Yaskawa INFORM job: A_NAIHAN_0617_1_PAINT_3.JBI

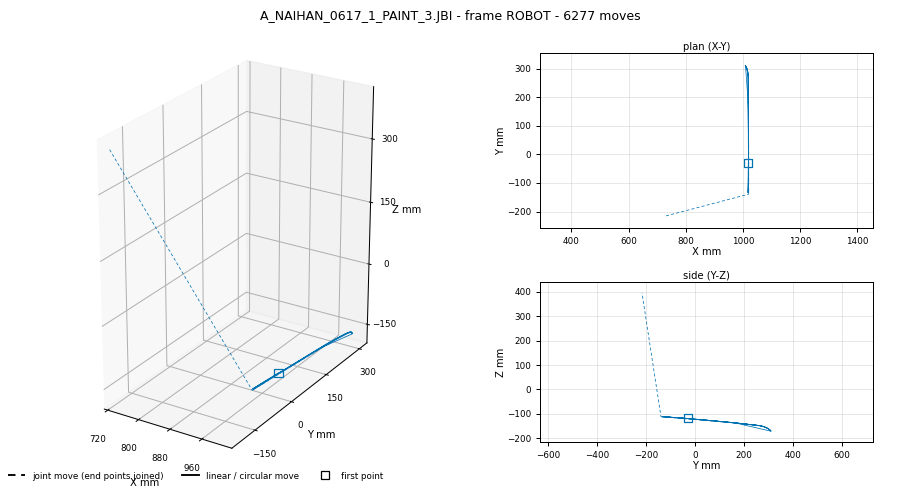
[picture p0: tool path of A_NAIHAN_0617_1_PAINT_3.JBI in frame ROBOT, 6277 of 6277 moves have a stored position in this frame; points joined in program order, loops and branches not executed]
/JOB
//NAME A_NAIHAN_0617_1_PAINT3
//POS
///NPOS 6277,0,0,0,0,0
///TOOL 1
///USER 0
///POSTYPE ROBOT
///RECTAN
///RCONF 0,0,0,0,1,0,0,0,0,0,0,0,0,0,0,0,0,0,0,0,0,0,0,0
C00000=1018.547,-30.236,-118.214,-24.117,21.565,-43.265
C00001=1018.547,-30.633,-118.183,-24.117,21.566,-43.271
C00002=1018.546,-31.031,-118.151,-24.116,21.567,-43.277
C00003=1018.545,-31.428,-118.119,-24.115,21.568,-43.282
C00004=1018.545,-31.825,-118.086,-24.114,21.567,-43.287
C00005=1018.543,-32.223,-118.054,-24.114,21.568,-43.293
C00006=1018.543,-32.621,-118.022,-24.113,21.569,-43.299
C00007=1018.542,-33.018,-117.990,-24.112,21.570,-43.304
C00008=1018.541,-33.415,-117.958,-24.111,21.570,-43.310
C00009=1018.540,-33.812,-117.926,-24.111,21.570,-43.315
C00010=1018.539,-34.210,-117.894,-24.110,21.571,-43.321
C00011=1018.539,-34.608,-117.863,-24.109,21.571,-43.328
C00012=1018.538,-35.005,-117.831,-24.108,21.572,-43.334
C00013=1018.536,-35.402,-117.799,-24.107,21.572,-43.339
C00014=1018.535,-35.799,-117.767,-24.107,21.573,-43.344
C00015=1018.535,-36.197,-117.735,-24.106,21.573,-43.350
C00016=1018.533,-36.594,-117.703,-24.105,21.574,-43.356
C00017=1018.532,-36.992,-117.671,-24.105,21.575,-43.361
C00018=1018.531,-37.389,-117.640,-24.104,21.575,-43.366
C00019=1018.530,-37.786,-117.608,-24.103,21.576,-43.372
C00020=1018.529,-38.183,-117.577,-24.102,21.576,-43.378
C00021=1018.528,-38.581,-117.544,-24.102,21.577,-43.383
C00022=1018.527,-38.978,-117.513,-24.101,21.578,-43.389
C00023=1018.526,-39.375,-117.481,-24.100,21.578,-43.394
C00024=1018.524,-39.772,-117.450,-24.099,21.579,-43.400
C00025=1018.524,-40.170,-117.418,-24.099,21.579,-43.405
C00026=1018.522,-40.567,-117.387,-24.098,21.580,-43.411
C00027=1018.520,-40.965,-117.355,-24.097,21.581,-43.417
C00028=1018.519,-41.362,-117.323,-24.096,21.582,-43.422
C00029=1018.518,-41.760,-117.292,-24.096,21.582,-43.427
C00030=1018.517,-42.156,-117.260,-24.095,21.582,-43.433
C00031=1018.515,-42.553,-117.228,-24.094,21.583,-43.439
C00032=1018.514,-42.951,-117.198,-24.093,21.584,-43.444
C00033=1018.513,-43.348,-117.166,-24.092,21.584,-43.451
C00034=1018.512,-43.745,-117.134,-24.092,21.585,-43.457
C00035=1018.511,-44.143,-117.103,-24.091,21.585,-43.462
C00036=1018.509,-44.540,-117.071,-24.090,21.585,-43.468
C00037=1018.508,-44.937,-117.040,-24.089,21.586,-43.473
C00038=1018.506,-45.334,-117.009,-24.089,21.587,-43.479
C00039=1018.505,-45.731,-116.977,-24.088,21.588,-43.485
C00040=1018.503,-46.128,-116.946,-24.087,21.589,-43.490
C00041=1018.501,-46.525,-116.915,-24.086,21.588,-43.496
C00042=1018.499,-46.923,-116.883,-24.086,21.589,-43.501
C00043=1018.498,-47.320,-116.853,-24.085,21.590,-43.507
C00044=1018.497,-47.717,-116.821,-24.084,21.591,-43.512
C00045=1018.496,-47.937,-116.804,-24.084,21.591,-43.516
C00046=1018.495,-48.156,-116.786,-24.083,21.591,-43.520
C00047=1018.493,-48.511,-116.759,-24.083,21.592,-43.525
C00048=1018.492,-48.908,-116.728,-24.082,21.592,-43.531
C00049=1018.490,-49.305,-116.696,-24.081,21.592,-43.536
C00050=1018.488,-49.703,-116.666,-24.080,21.593,-43.542
C00051=1018.487,-50.099,-116.634,-24.080,21.594,-43.547
C00052=1018.485,-50.496,-116.603,-24.079,21.595,-43.553
C00053=1018.483,-50.894,-116.572,-24.078,21.595,-43.558
C00054=1018.482,-51.291,-116.541,-24.077,21.596,-43.564
C00055=1018.479,-51.687,-116.510,-24.077,21.597,-43.570
C00056=1018.478,-52.085,-116.479,-24.076,21.598,-43.575
C00057=1018.477,-52.481,-116.448,-24.075,21.598,-43.581
C00058=1018.474,-52.877,-116.417,-24.074,21.598,-43.588
C00059=1018.473,-53.275,-116.386,-24.073,21.599,-43.593
C00060=1018.471,-53.671,-116.355,-24.073,21.599,-43.599
C00061=1018.469,-54.068,-116.324,-24.072,21.600,-43.604
C00062=1018.467,-54.466,-116.293,-24.071,21.601,-43.610
C00063=1018.465,-54.862,-116.262,-24.071,21.602,-43.616
C00064=1018.463,-55.259,-116.232,-24.070,21.603,-43.621
C00065=1018.461,-55.657,-116.200,-24.069,21.602,-43.627
C00066=1018.459,-56.054,-116.170,-24.068,21.603,-43.632
C00067=1018.457,-56.452,-116.139,-24.067,21.603,-43.639
C00068=1018.455,-56.850,-116.108,-24.067,21.604,-43.645
C00069=1018.452,-57.248,-116.077,-24.066,21.605,-43.651
C00070=1018.451,-57.647,-116.047,-24.065,21.606,-43.656
C00071=1018.449,-58.047,-116.016,-24.064,21.606,-43.662
C00072=1018.447,-58.447,-115.985,-24.064,21.607,-43.667
C00073=1018.445,-58.846,-115.954,-24.063,21.608,-43.673
C00074=1018.443,-59.247,-115.923,-24.062,21.608,-43.680
C00075=1018.441,-59.648,-115.892,-24.061,21.609,-43.686
C00076=1018.438,-60.050,-115.861,-24.061,21.610,-43.691
C00077=1018.436,-60.453,-115.831,-24.060,21.610,-43.697
C00078=1018.434,-60.856,-115.799,-24.059,21.610,-43.702
C00079=1018.431,-61.260,-115.768,-24.058,21.611,-43.708
C00080=1018.429,-61.663,-115.737,-24.057,21.611,-43.715
C00081=1018.427,-62.068,-115.705,-24.057,21.612,-43.720
C00082=1018.424,-62.473,-115.675,-24.056,21.613,-43.726
C00083=1018.421,-62.879,-115.643,-24.055,21.614,-43.732
C00084=1018.419,-63.285,-115.612,-24.054,21.615,-43.737
C00085=1018.417,-63.691,-115.581,-24.053,21.615,-43.744
C00086=1018.415,-64.099,-115.550,-24.053,21.615,-43.750
C00087=1018.412,-64.506,-115.519,-24.052,21.616,-43.756
C00088=1018.409,-64.915,-115.487,-24.051,21.617,-43.761
C00089=1018.407,-65.323,-115.457,-24.050,21.617,-43.768
C00090=1018.404,-65.732,-115.425,-24.049,21.618,-43.774
C00091=1018.402,-66.142,-115.394,-24.049,21.619,-43.780
C00092=1018.399,-66.551,-115.362,-24.048,21.620,-43.785
C00093=1018.396,-66.961,-115.331,-24.047,21.620,-43.791
C00094=1018.393,-67.371,-115.300,-24.046,21.621,-43.798
C00095=1018.391,-67.781,-115.269,-24.046,21.621,-43.804
C00096=1018.388,-68.191,-115.238,-24.045,21.622,-43.809
C00097=1018.385,-68.601,-115.206,-24.044,21.623,-43.815
C00098=1018.382,-69.013,-115.175,-24.043,21.623,-43.822
C00099=1018.380,-69.423,-115.144,-24.042,21.624,-43.827
C00100=1018.377,-69.834,-115.113,-24.042,21.625,-43.833
C00101=1018.374,-70.245,-115.082,-24.041,21.625,-43.839
C00102=1018.371,-70.656,-115.050,-24.040,21.626,-43.846
C00103=1018.368,-71.067,-115.019,-24.039,21.626,-43.851
C00104=1018.365,-71.478,-114.989,-24.039,21.627,-43.857
C00105=1018.362,-71.888,-114.957,-24.038,21.628,-43.865
C00106=1018.359,-72.299,-114.926,-24.037,21.629,-43.870
C00107=1018.356,-72.710,-114.895,-24.036,21.630,-43.876
C00108=1018.353,-73.121,-114.864,-24.035,21.631,-43.881
C00109=1018.350,-73.532,-114.833,-24.034,21.631,-43.888
C00110=1018.348,-73.942,-114.803,-24.034,21.632,-43.894
C00111=1018.344,-74.353,-114.771,-24.033,21.632,-43.900
C00112=1018.341,-74.763,-114.740,-24.032,21.633,-43.905
C00113=1018.338,-75.173,-114.710,-24.031,21.633,-43.912
C00114=1018.335,-75.583,-114.679,-24.031,21.634,-43.918
C00115=1018.331,-75.993,-114.648,-24.030,21.635,-43.924
C00116=1018.329,-76.402,-114.617,-24.029,21.636,-43.929
C00117=1018.326,-76.810,-114.586,-24.028,21.636,-43.936
C00118=1018.321,-77.220,-114.556,-24.027,21.637,-43.942
C00119=1018.319,-77.628,-114.525,-24.027,21.637,-43.948
C00120=1018.315,-78.036,-114.494,-24.026,21.638,-43.953
C00121=1018.312,-78.443,-114.464,-24.025,21.638,-43.960
C00122=1018.309,-78.851,-114.434,-24.024,21.639,-43.966
C00123=1018.305,-79.257,-114.403,-24.023,21.640,-43.972
C00124=1018.302,-79.663,-114.373,-24.023,21.641,-43.977
C00125=1018.299,-80.069,-114.342,-24.022,21.641,-43.984
C00126=1018.295,-80.474,-114.313,-24.021,21.642,-43.990
C00127=1018.292,-80.878,-114.283,-24.020,21.643,-43.995
C00128=1018.288,-81.283,-114.252,-24.020,21.643,-44.001
C00129=1018.285,-81.686,-114.222,-24.019,21.644,-44.007
C00130=1018.281,-82.089,-114.192,-24.018,21.644,-44.014
C00131=1018.278,-82.490,-114.162,-24.017,21.645,-44.019
C00132=1018.274,-82.892,-114.133,-24.016,21.646,-44.025
C00133=1018.271,-83.293,-114.103,-24.016,21.647,-44.031
C00134=1018.267,-83.693,-114.073,-24.015,21.648,-44.036
C00135=1018.264,-84.093,-114.043,-24.014,21.648,-44.043
C00136=1018.260,-84.499,-114.013,-24.013,21.649,-44.049
C00137=1018.258,-84.723,-113.996,-24.013,21.649,-44.053
C00138=1018.256,-84.964,-113.979,-24.012,21.650,-44.056
C00139=1018.254,-85.218,-113.959,-24.012,21.649,-44.060
C00140=1018.251,-85.472,-113.941,-24.012,21.650,-44.062
C00141=1018.248,-85.718,-113.923,-24.011,21.650,-44.065
C00142=1018.246,-85.948,-113.905,-24.011,21.651,-44.069
C00143=1018.243,-86.357,-113.875,-24.010,21.652,-44.077
C00144=1018.239,-86.745,-113.846,-24.009,21.652,-44.082
C00145=1018.236,-87.125,-113.818,-24.008,21.652,-44.087
C00146=1018.232,-87.497,-113.791,-24.007,21.653,-44.093
C00147=1018.228,-87.869,-113.764,-24.007,21.654,-44.099
C00148=1018.225,-88.244,-113.736,-24.006,21.655,-44.104
C00149=1018.221,-88.652,-113.706,-24.005,21.656,-44.112
C00150=1018.218,-88.899,-113.688,-24.005,21.656,-44.116
C00151=1018.216,-89.174,-113.668,-24.004,21.657,-44.117
C00152=1018.213,-89.458,-113.646,-24.004,21.656,-44.121
C00153=1018.210,-89.733,-113.626,-24.003,21.657,-44.124
C00154=1018.208,-89.983,-113.607,-24.003,21.657,-44.128
C00155=1018.205,-90.202,-113.591,-24.002,21.658,-44.132
C00156=1018.201,-90.598,-113.563,-24.002,21.659,-44.138
C00157=1018.198,-90.992,-113.534,-24.001,21.659,-44.145
C00158=1018.194,-91.384,-113.505,-24.000,21.660,-44.150
C00159=1018.190,-91.776,-113.476,-23.999,21.660,-44.156
C00160=1018.186,-92.168,-113.447,-23.999,21.661,-44.162
C00161=1018.182,-92.558,-113.419,-23.998,21.662,-44.167
C00162=1018.178,-92.948,-113.390,-23.997,21.663,-44.173
C00163=1018.174,-93.338,-113.362,-23.996,21.664,-44.178
C00164=1018.170,-93.726,-113.333,-23.996,21.664,-44.184
C00165=1018.166,-94.113,-113.305,-23.995,21.664,-44.189
C00166=1018.162,-94.500,-113.277,-23.994,21.665,-44.195
C00167=1018.157,-94.886,-113.248,-23.994,21.666,-44.200
C00168=1018.153,-95.272,-113.220,-23.993,21.666,-44.207
C00169=1018.149,-95.657,-113.192,-23.992,21.667,-44.213
C00170=1018.145,-96.041,-113.164,-23.991,21.668,-44.219
C00171=1018.141,-96.425,-113.136,-23.990,21.668,-44.224
C00172=1018.136,-96.809,-113.109,-23.990,21.669,-44.230
C00173=1018.132,-97.193,-113.081,-23.989,21.669,-44.235
C00174=1018.127,-97.576,-113.053,-23.988,21.670,-44.241
C00175=1018.124,-97.959,-113.025,-23.988,21.671,-44.246
C00176=1018.119,-98.342,-112.997,-23.987,21.672,-44.252
C00177=1018.116,-98.726,-112.969,-23.986,21.673,-44.258
C00178=1018.111,-99.109,-112.941,-23.985,21.673,-44.263
C00179=1018.106,-99.493,-112.914,-23.985,21.673,-44.268
C00180=1018.102,-99.877,-112.885,-23.984,21.674,-44.274
C00181=1018.097,-100.261,-112.857,-23.983,21.675,-44.280
C00182=1018.093,-100.647,-112.830,-23.982,21.676,-44.285
C00183=1018.089,-101.032,-112.802,-23.982,21.677,-44.291
C00184=1018.084,-101.418,-112.774,-23.981,21.676,-44.296
C00185=1018.079,-101.806,-112.746,-23.980,21.677,-44.302
C00186=1018.075,-102.194,-112.718,-23.980,21.678,-44.307
C00187=1018.070,-102.582,-112.690,-23.979,21.678,-44.314
C00188=1018.065,-102.971,-112.661,-23.978,21.679,-44.320
C00189=1018.060,-103.361,-112.634,-23.977,21.680,-44.326
C00190=1018.056,-103.751,-112.606,-23.976,21.681,-44.331
C00191=1018.051,-104.143,-112.577,-23.976,21.682,-44.337
C00192=1018.046,-104.535,-112.549,-23.975,21.681,-44.342
C00193=1018.041,-104.926,-112.521,-23.974,21.682,-44.348
C00194=1018.037,-105.318,-112.492,-23.974,21.683,-44.353
C00195=1018.032,-105.711,-112.464,-23.973,21.684,-44.359
C00196=1018.027,-106.104,-112.436,-23.972,21.685,-44.365
C00197=1018.022,-106.497,-112.408,-23.971,21.686,-44.370
C00198=1018.017,-106.890,-112.380,-23.971,21.686,-44.376
C00199=1018.012,-107.283,-112.352,-23.970,21.687,-44.383
C00200=1018.006,-107.675,-112.323,-23.969,21.687,-44.388
C00201=1018.002,-108.068,-112.295,-23.968,21.688,-44.394
C00202=1017.997,-108.461,-112.267,-23.968,21.688,-44.399
C00203=1017.992,-108.854,-112.239,-23.967,21.689,-44.405
C00204=1017.986,-109.247,-112.211,-23.966,21.690,-44.411
C00205=1017.981,-109.639,-112.183,-23.965,21.691,-44.416
C00206=1017.976,-110.032,-112.155,-23.965,21.691,-44.422
C00207=1017.971,-110.425,-112.127,-23.964,21.692,-44.427
C00208=1017.966,-110.818,-112.099,-23.963,21.693,-44.433
C00209=1017.961,-111.211,-112.071,-23.963,21.694,-44.439
C00210=1017.954,-111.603,-112.043,-23.962,21.694,-44.446
C00211=1017.949,-111.996,-112.015,-23.961,21.694,-44.451
C00212=1017.944,-112.389,-111.987,-23.960,21.695,-44.456
C00213=1017.938,-112.781,-111.958,-23.959,21.696,-44.462
C00214=1017.933,-113.174,-111.930,-23.959,21.696,-44.468
C00215=1017.927,-113.567,-111.903,-23.958,21.697,-44.473
C00216=1017.922,-113.959,-111.874,-23.957,21.698,-44.479
C00217=1017.916,-114.352,-111.847,-23.957,21.699,-44.485
C00218=1017.911,-114.745,-111.819,-23.956,21.700,-44.490
C00219=1017.906,-115.136,-111.791,-23.955,21.701,-44.496
C00220=1017.900,-115.529,-111.764,-23.954,21.700,-44.501
C00221=1017.894,-115.921,-111.735,-23.954,21.701,-44.507
C00222=1017.889,-116.314,-111.708,-23.953,21.702,-44.512
C00223=1017.883,-116.706,-111.680,-23.952,21.703,-44.518
C00224=1017.877,-117.099,-111.652,-23.952,21.704,-44.523
C00225=1017.872,-117.492,-111.624,-23.951,21.705,-44.529
C00226=1017.866,-117.883,-111.596,-23.950,21.705,-44.536
C00227=1017.860,-118.276,-111.569,-23.949,21.705,-44.541
C00228=1017.854,-118.668,-111.541,-23.948,21.706,-44.547
C00229=1017.849,-119.060,-111.513,-23.948,21.706,-44.553
C00230=1017.842,-119.452,-111.485,-23.947,21.707,-44.558
C00231=1017.837,-119.845,-111.458,-23.946,21.708,-44.564
C00232=1017.831,-120.237,-111.430,-23.946,21.709,-44.569
C00233=1017.824,-120.628,-111.403,-23.945,21.710,-44.575
C00234=1017.819,-121.021,-111.375,-23.944,21.710,-44.580
C00235=1017.812,-121.413,-111.347,-23.943,21.710,-44.586
C00236=1017.807,-121.805,-111.320,-23.943,21.711,-44.591
C00237=1017.800,-122.197,-111.292,-23.942,21.712,-44.597
C00238=1017.794,-122.590,-111.265,-23.941,21.713,-44.603
C00239=1017.788,-122.982,-111.237,-23.941,21.714,-44.608
C00240=1017.782,-123.373,-111.209,-23.940,21.715,-44.614
C00241=1017.776,-123.766,-111.182,-23.939,21.714,-44.619
C00242=1017.770,-124.158,-111.154,-23.939,21.715,-44.625
C00243=1017.763,-124.549,-111.126,-23.938,21.716,-44.630
C00244=1017.757,-124.942,-111.099,-23.937,21.717,-44.636
C00245=1017.750,-125.334,-111.072,-23.936,21.718,-44.642
C00246=1017.743,-125.725,-111.044,-23.936,21.719,-44.647
C00247=1017.738,-126.117,-111.017,-23.935,21.719,-44.652
C00248=1017.731,-126.509,-110.989,-23.934,21.719,-44.658
C00249=1017.725,-126.901,-110.962,-23.934,21.720,-44.664
C00250=1017.719,-127.294,-110.934,-23.933,21.721,-44.669
C00251=1017.712,-127.685,-110.907,-23.932,21.722,-44.675
C00252=1017.705,-128.077,-110.879,-23.932,21.723,-44.680
C00253=1017.699,-128.469,-110.853,-23.931,21.723,-44.686
C00254=1017.692,-128.861,-110.825,-23.930,21.723,-44.691
C00255=1017.685,-129.253,-110.798,-23.929,21.724,-44.697
C00256=1017.679,-129.644,-110.770,-23.929,21.725,-44.703
C00257=1017.672,-130.036,-110.744,-23.928,21.726,-44.708
C00258=1017.665,-130.428,-110.716,-23.927,21.727,-44.714
C00259=1017.658,-130.820,-110.689,-23.926,21.727,-44.719
C00260=1017.652,-131.211,-110.661,-23.926,21.728,-44.725
C00261=1017.645,-131.604,-110.634,-23.925,21.728,-44.730
C00262=1017.638,-131.995,-110.607,-23.924,21.729,-44.736
C00263=1017.631,-132.387,-110.579,-23.924,21.730,-44.741
C00264=1017.625,-132.779,-110.552,-23.923,21.730,-44.747
C00265=1017.618,-133.171,-110.524,-23.922,21.731,-44.752
C00266=1017.610,-133.563,-110.498,-23.922,21.732,-44.758
C00267=1017.604,-133.954,-110.470,-23.921,21.732,-44.763
C00268=1017.988,-133.926,-110.710,-23.921,21.732,-44.763
C00269=1017.995,-133.535,-110.737,-23.922,21.732,-44.758
C00270=1018.002,-133.143,-110.765,-23.922,21.731,-44.752
C00271=1018.008,-132.751,-110.792,-23.923,21.730,-44.747
C00272=1018.015,-132.360,-110.818,-23.924,21.730,-44.741
C00273=1018.022,-131.968,-110.846,-23.924,21.729,-44.736
C00274=1018.029,-131.576,-110.872,-23.925,21.728,-44.730
C00275=1018.035,-131.184,-110.900,-23.926,21.728,-44.725
C00276=1018.042,-130.792,-110.928,-23.926,21.727,-44.719
C00277=1018.049,-130.400,-110.954,-23.927,21.727,-44.714
C00278=1018.055,-130.009,-110.982,-23.928,21.726,-44.708
C00279=1018.062,-129.617,-111.009,-23.929,21.725,-44.703
C00280=1018.068,-129.225,-111.036,-23.929,21.724,-44.697
C00281=1018.075,-128.833,-111.064,-23.930,21.723,-44.691
C00282=1018.081,-128.441,-111.091,-23.931,21.723,-44.686
C00283=1018.087,-128.050,-111.118,-23.932,21.723,-44.680
C00284=1018.094,-127.658,-111.145,-23.932,21.722,-44.675
C00285=1018.101,-127.265,-111.172,-23.933,21.721,-44.669
C00286=1018.107,-126.873,-111.200,-23.934,21.720,-44.664
C00287=1018.113,-126.482,-111.227,-23.934,21.719,-44.658
C00288=1018.120,-126.090,-111.254,-23.935,21.719,-44.652
C00289=1018.126,-125.698,-111.283,-23.936,21.719,-44.647
C00290=1018.132,-125.306,-111.309,-23.936,21.718,-44.642
C00291=1018.138,-124.914,-111.337,-23.937,21.717,-44.636
C00292=1018.144,-124.522,-111.364,-23.938,21.716,-44.630
C00293=1018.150,-124.130,-111.392,-23.939,21.715,-44.625
C00294=1018.157,-123.738,-111.419,-23.939,21.714,-44.619
C00295=1018.162,-123.346,-111.447,-23.940,21.715,-44.614
C00296=1018.168,-122.954,-111.474,-23.941,21.714,-44.608
C00297=1018.175,-122.562,-111.502,-23.941,21.713,-44.603
C00298=1018.180,-122.170,-111.529,-23.942,21.712,-44.597
C00299=1018.186,-121.778,-111.557,-23.943,21.711,-44.591
C00300=1018.192,-121.385,-111.584,-23.943,21.710,-44.586
C00301=1018.198,-120.993,-111.612,-23.944,21.710,-44.580
C00302=1018.204,-120.602,-111.639,-23.945,21.710,-44.575
C00303=1018.210,-120.210,-111.667,-23.946,21.709,-44.569
C00304=1018.216,-119.817,-111.694,-23.946,21.708,-44.564
C00305=1018.222,-119.425,-111.722,-23.947,21.707,-44.558
C00306=1018.227,-119.033,-111.749,-23.948,21.706,-44.553
C00307=1018.233,-118.641,-111.777,-23.948,21.706,-44.547
C00308=1018.239,-118.248,-111.805,-23.949,21.705,-44.541
C00309=1018.244,-117.855,-111.833,-23.950,21.705,-44.536
C00310=1018.250,-117.464,-111.861,-23.951,21.705,-44.529
C00311=1018.256,-117.071,-111.888,-23.952,21.704,-44.523
C00312=1018.261,-116.679,-111.915,-23.952,21.703,-44.518
C00313=1018.267,-116.287,-111.944,-23.953,21.702,-44.512
C00314=1018.272,-115.894,-111.971,-23.954,21.701,-44.507
C00315=1018.278,-115.502,-111.999,-23.954,21.700,-44.501
C00316=1018.284,-115.110,-112.027,-23.955,21.701,-44.496
C00317=1018.289,-114.717,-112.055,-23.956,21.700,-44.490
C00318=1018.294,-114.325,-112.082,-23.957,21.699,-44.485
C00319=1018.299,-113.932,-112.110,-23.957,21.698,-44.479
C00320=1018.305,-113.540,-112.138,-23.958,21.697,-44.473
C00321=1018.310,-113.147,-112.166,-23.959,21.696,-44.468
C00322=1018.316,-112.755,-112.194,-23.959,21.696,-44.462
C00323=1018.321,-112.362,-112.222,-23.960,21.695,-44.456
C00324=1018.326,-111.969,-112.250,-23.961,21.694,-44.451
C00325=1018.332,-111.577,-112.277,-23.962,21.694,-44.446
C00326=1018.337,-111.184,-112.305,-23.963,21.694,-44.439
C00327=1018.342,-110.791,-112.334,-23.963,21.693,-44.433
C00328=1018.347,-110.398,-112.362,-23.964,21.692,-44.427
C00329=1018.352,-110.005,-112.390,-23.965,21.691,-44.422
C00330=1018.357,-109.612,-112.418,-23.965,21.691,-44.416
C00331=1018.362,-109.219,-112.446,-23.966,21.690,-44.411
C00332=1018.367,-108.827,-112.473,-23.967,21.689,-44.405
C00333=1018.372,-108.434,-112.501,-23.968,21.688,-44.399
C00334=1018.377,-108.041,-112.529,-23.968,21.688,-44.394
C00335=1018.382,-107.649,-112.558,-23.969,21.687,-44.388
C00336=1018.387,-107.256,-112.586,-23.970,21.687,-44.383
C00337=1018.392,-106.863,-112.614,-23.971,21.686,-44.376
C00338=1018.397,-106.470,-112.642,-23.971,21.686,-44.370
C00339=1018.402,-106.077,-112.670,-23.972,21.685,-44.365
C00340=1018.407,-105.684,-112.699,-23.973,21.684,-44.359
C00341=1018.412,-105.291,-112.727,-23.974,21.683,-44.353
C00342=1018.417,-104.899,-112.755,-23.974,21.682,-44.348
C00343=1018.421,-104.507,-112.783,-23.975,21.681,-44.342
C00344=1018.426,-104.115,-112.811,-23.976,21.682,-44.337
C00345=1018.430,-103.724,-112.839,-23.976,21.681,-44.331
C00346=1018.435,-103.334,-112.867,-23.977,21.680,-44.326
C00347=1018.440,-102.944,-112.895,-23.978,21.679,-44.320
C00348=1018.444,-102.555,-112.924,-23.979,21.678,-44.314
C00349=1018.449,-102.167,-112.952,-23.980,21.678,-44.307
C00350=1018.454,-101.779,-112.979,-23.980,21.677,-44.302
C00351=1018.458,-101.391,-113.007,-23.981,21.676,-44.296
C00352=1018.463,-101.005,-113.035,-23.982,21.677,-44.291
C00353=1018.467,-100.620,-113.063,-23.982,21.676,-44.285
C00354=1018.471,-100.234,-113.091,-23.983,21.675,-44.280
C00355=1018.476,-99.849,-113.119,-23.984,21.674,-44.274
C00356=1018.480,-99.465,-113.146,-23.985,21.673,-44.268
C00357=1018.485,-99.082,-113.175,-23.985,21.673,-44.263
C00358=1018.489,-98.699,-113.202,-23.986,21.673,-44.258
C00359=1018.493,-98.315,-113.230,-23.987,21.672,-44.252
C00360=1018.497,-97.932,-113.258,-23.988,21.671,-44.246
C00361=1018.500,-97.617,-113.280,-23.988,21.670,-44.241
C00362=1018.503,-97.391,-113.297,-23.988,21.670,-44.239
C00363=1018.505,-97.166,-113.313,-23.989,21.669,-44.235
C00364=1018.510,-96.782,-113.342,-23.990,21.669,-44.230
C00365=1018.514,-96.398,-113.369,-23.990,21.668,-44.224
C00366=1018.518,-96.014,-113.397,-23.991,21.668,-44.219
C00367=1018.522,-95.630,-113.424,-23.992,21.667,-44.213
C00368=1018.526,-95.245,-113.453,-23.993,21.666,-44.207
C00369=1018.530,-94.860,-113.481,-23.994,21.666,-44.200
C00370=1018.534,-94.473,-113.510,-23.994,21.665,-44.195
C00371=1018.539,-94.086,-113.537,-23.995,21.664,-44.189
C00372=1018.543,-93.698,-113.566,-23.996,21.664,-44.184
C00373=1018.547,-93.310,-113.594,-23.996,21.664,-44.178
C00374=1018.551,-92.921,-113.623,-23.997,21.663,-44.173
C00375=1018.555,-92.531,-113.651,-23.998,21.662,-44.167
C00376=1018.558,-92.140,-113.680,-23.999,21.661,-44.162
C00377=1018.562,-91.749,-113.708,-23.999,21.660,-44.156
C00378=1018.566,-91.357,-113.737,-24.000,21.660,-44.150
C00379=1018.570,-90.964,-113.766,-24.001,21.659,-44.145
C00380=1018.574,-90.570,-113.794,-24.002,21.659,-44.138
C00381=1018.578,-90.174,-113.824,-24.002,21.658,-44.132
C00382=1018.580,-89.956,-113.840,-24.003,21.657,-44.128
C00383=1018.582,-89.706,-113.858,-24.003,21.657,-44.124
C00384=1018.585,-89.431,-113.879,-24.004,21.656,-44.121
C00385=1018.588,-89.147,-113.900,-24.004,21.657,-44.117
C00386=1018.591,-88.872,-113.919,-24.005,21.656,-44.116
C00387=1018.592,-88.625,-113.938,-24.005,21.656,-44.112
C00388=1018.597,-88.218,-113.968,-24.006,21.655,-44.104
C00389=1018.600,-87.842,-113.996,-24.007,21.654,-44.099
C00390=1018.603,-87.470,-114.023,-24.007,21.653,-44.093
C00391=1018.607,-87.098,-114.050,-24.008,21.652,-44.087
C00392=1018.610,-86.719,-114.078,-24.009,21.652,-44.082
C00393=1018.614,-86.330,-114.107,-24.010,21.652,-44.077
C00394=1018.618,-85.921,-114.137,-24.011,21.651,-44.069
C00395=1018.620,-85.691,-114.154,-24.011,21.650,-44.065
C00396=1018.622,-85.445,-114.172,-24.012,21.650,-44.062
C00397=1018.625,-85.190,-114.191,-24.012,21.649,-44.060
C00398=1018.627,-84.937,-114.210,-24.012,21.650,-44.056
C00399=1018.629,-84.696,-114.228,-24.013,21.649,-44.053
C00400=1018.631,-84.472,-114.244,-24.013,21.649,-44.049
C00401=1018.635,-84.066,-114.275,-24.014,21.648,-44.043
C00402=1018.638,-83.666,-114.303,-24.015,21.648,-44.036
C00403=1018.642,-83.266,-114.333,-24.016,21.647,-44.031
C00404=1018.645,-82.865,-114.363,-24.016,21.646,-44.025
C00405=1018.648,-82.464,-114.394,-24.017,21.645,-44.019
C00406=1018.652,-82.062,-114.423,-24.018,21.644,-44.014
C00407=1018.656,-81.659,-114.453,-24.019,21.644,-44.007
C00408=1018.659,-81.256,-114.483,-24.020,21.643,-44.001
C00409=1018.662,-80.851,-114.513,-24.020,21.643,-43.995
C00410=1018.665,-80.448,-114.543,-24.021,21.642,-43.990
C00411=1018.669,-80.042,-114.573,-24.022,21.641,-43.984
C00412=1018.673,-79.637,-114.604,-24.023,21.641,-43.977
C00413=1018.675,-79.230,-114.634,-24.023,21.640,-43.972
C00414=1018.679,-78.824,-114.664,-24.024,21.639,-43.966
C00415=1018.682,-78.417,-114.695,-24.025,21.638,-43.960
C00416=1018.685,-78.009,-114.725,-24.026,21.638,-43.953
C00417=1018.689,-77.601,-114.756,-24.027,21.637,-43.948
C00418=1018.692,-77.193,-114.787,-24.027,21.637,-43.942
C00419=1018.695,-76.784,-114.817,-24.028,21.636,-43.936
C00420=1018.698,-76.375,-114.848,-24.029,21.636,-43.929
C00421=1018.702,-75.966,-114.879,-24.030,21.635,-43.924
C00422=1018.705,-75.557,-114.909,-24.031,21.634,-43.918
C00423=1018.707,-75.146,-114.940,-24.031,21.633,-43.912
C00424=1018.711,-74.736,-114.971,-24.032,21.633,-43.905
C00425=1018.714,-74.326,-115.002,-24.033,21.632,-43.900
C00426=1018.717,-73.915,-115.032,-24.034,21.632,-43.894
C00427=1018.720,-73.505,-115.064,-24.034,21.631,-43.888
C00428=1018.723,-73.095,-115.094,-24.035,21.631,-43.881
C00429=1018.726,-72.683,-115.125,-24.036,21.630,-43.876
C00430=1018.729,-72.273,-115.157,-24.037,21.629,-43.870
C00431=1018.732,-71.862,-115.187,-24.038,21.628,-43.865
C00432=1018.735,-71.451,-115.218,-24.039,21.627,-43.857
C00433=1018.738,-71.041,-115.250,-24.039,21.626,-43.851
C00434=1018.741,-70.629,-115.281,-24.040,21.626,-43.846
C00435=1018.743,-70.218,-115.312,-24.041,21.625,-43.839
C00436=1018.746,-69.807,-115.343,-24.042,21.625,-43.833
C00437=1018.749,-69.397,-115.374,-24.042,21.624,-43.827
C00438=1018.752,-68.986,-115.405,-24.043,21.623,-43.822
C00439=1018.755,-68.576,-115.437,-24.044,21.623,-43.815
C00440=1018.757,-68.164,-115.468,-24.045,21.622,-43.809
C00441=1018.760,-67.754,-115.499,-24.046,21.621,-43.804
C00442=1018.763,-67.344,-115.531,-24.046,21.621,-43.798
C00443=1018.764,-66.934,-115.561,-24.047,21.620,-43.791
C00444=1018.767,-66.524,-115.592,-24.048,21.620,-43.785
C00445=1018.770,-66.115,-115.624,-24.049,21.619,-43.780
C00446=1018.773,-65.705,-115.655,-24.049,21.618,-43.774
C00447=1018.776,-65.297,-115.686,-24.050,21.617,-43.768
C00448=1018.778,-64.888,-115.717,-24.051,21.617,-43.761
C00449=1018.780,-64.480,-115.749,-24.052,21.616,-43.756
C00450=1018.783,-64.073,-115.780,-24.053,21.615,-43.750
C00451=1018.785,-63.666,-115.810,-24.053,21.615,-43.744
C00452=1018.787,-63.258,-115.842,-24.054,21.615,-43.737
C00453=1018.790,-62.852,-115.873,-24.055,21.614,-43.732
C00454=1018.793,-62.447,-115.904,-24.056,21.613,-43.726
C00455=1018.795,-62.041,-115.935,-24.057,21.612,-43.720
C00456=1018.796,-61.637,-115.966,-24.057,21.611,-43.715
C00457=1018.800,-61.233,-115.998,-24.058,21.611,-43.708
C00458=1018.802,-60.829,-116.028,-24.059,21.610,-43.702
C00459=1018.804,-60.426,-116.059,-24.060,21.610,-43.697
C00460=1018.806,-60.024,-116.091,-24.061,21.610,-43.691
C00461=1018.808,-59.622,-116.121,-24.061,21.609,-43.686
C00462=1018.810,-59.221,-116.152,-24.062,21.608,-43.680
C00463=1018.812,-58.820,-116.184,-24.063,21.608,-43.673
C00464=1018.815,-58.419,-116.214,-24.064,21.607,-43.667
C00465=1018.817,-58.020,-116.245,-24.064,21.606,-43.662
C00466=1018.818,-57.621,-116.276,-24.065,21.606,-43.656
C00467=1018.821,-57.222,-116.307,-24.066,21.605,-43.651
C00468=1018.823,-56.824,-116.338,-24.067,21.604,-43.645
C00469=1018.825,-56.425,-116.369,-24.067,21.603,-43.639
C00470=1018.827,-56.028,-116.399,-24.068,21.603,-43.632
C00471=1018.829,-55.630,-116.430,-24.069,21.602,-43.627
C00472=1018.831,-55.233,-116.461,-24.070,21.603,-43.621
C00473=1018.833,-54.836,-116.492,-24.071,21.602,-43.616
C00474=1018.835,-54.439,-116.522,-24.071,21.601,-43.610
C00475=1018.836,-54.042,-116.554,-24.072,21.600,-43.604
C00476=1018.838,-53.645,-116.584,-24.073,21.599,-43.599
C00477=1018.841,-53.248,-116.615,-24.073,21.599,-43.593
C00478=1018.842,-52.851,-116.647,-24.074,21.598,-43.588
C00479=1018.844,-52.454,-116.677,-24.075,21.598,-43.581
C00480=1018.846,-52.057,-116.708,-24.076,21.598,-43.575
C00481=1018.847,-51.661,-116.739,-24.077,21.597,-43.570
C00482=1018.849,-51.264,-116.770,-24.077,21.596,-43.564
C00483=1018.851,-50.867,-116.801,-24.078,21.595,-43.558
C00484=1018.853,-50.470,-116.832,-24.079,21.595,-43.553
C00485=1018.854,-50.073,-116.863,-24.080,21.594,-43.547
C00486=1018.856,-49.676,-116.895,-24.080,21.593,-43.542
C00487=1018.858,-49.279,-116.925,-24.081,21.592,-43.536
C00488=1018.859,-48.882,-116.956,-24.082,21.592,-43.531
C00489=1018.861,-48.485,-116.988,-24.083,21.592,-43.525
C00490=1018.862,-48.087,-117.019,-24.084,21.592,-43.518
C00491=1018.864,-47.691,-117.050,-24.084,21.591,-43.512
C00492=1018.866,-47.294,-117.081,-24.085,21.590,-43.507
C00493=1018.867,-46.896,-117.112,-24.086,21.589,-43.501
C00494=1018.868,-46.499,-117.144,-24.086,21.588,-43.496
C00495=1018.869,-46.102,-117.175,-24.087,21.589,-43.490
C00496=1018.871,-45.705,-117.206,-24.088,21.588,-43.485
C00497=1018.872,-45.308,-117.238,-24.089,21.587,-43.479
C00498=1018.874,-44.910,-117.269,-24.089,21.586,-43.473
C00499=1018.875,-44.513,-117.300,-24.090,21.585,-43.468
C00500=1018.877,-44.116,-117.332,-24.091,21.585,-43.462
C00501=1018.878,-43.718,-117.363,-24.092,21.585,-43.457
C00502=1018.880,-43.321,-117.395,-24.092,21.584,-43.451
C00503=1018.881,-42.924,-117.426,-24.093,21.584,-43.444
C00504=1018.883,-42.527,-117.457,-24.094,21.583,-43.439
C00505=1018.884,-42.130,-117.489,-24.095,21.582,-43.433
C00506=1018.885,-41.733,-117.521,-24.096,21.582,-43.427
C00507=1018.886,-41.335,-117.552,-24.096,21.582,-43.422
C00508=1018.888,-40.938,-117.584,-24.097,21.581,-43.417
C00509=1018.889,-40.541,-117.615,-24.098,21.580,-43.411
C00510=1018.890,-40.143,-117.647,-24.099,21.579,-43.405
C00511=1018.891,-39.746,-117.678,-24.099,21.579,-43.400
C00512=1018.892,-39.349,-117.710,-24.100,21.578,-43.394
C00513=1018.893,-38.952,-117.741,-24.101,21.578,-43.389
C00514=1018.895,-38.555,-117.773,-24.102,21.577,-43.383
C00515=1018.895,-38.157,-117.805,-24.102,21.576,-43.378
C00516=1018.897,-37.760,-117.836,-24.103,21.576,-43.372
C00517=1018.898,-37.362,-117.868,-24.104,21.575,-43.366
C00518=1018.900,-36.965,-117.900,-24.105,21.575,-43.361
C00519=1018.900,-36.568,-117.932,-24.105,21.574,-43.356
C00520=1018.901,-36.170,-117.964,-24.106,21.573,-43.350
C00521=1018.902,-35.773,-117.995,-24.107,21.573,-43.344
C00522=1018.903,-35.376,-118.027,-24.107,21.572,-43.339
C00523=1018.903,-34.978,-118.059,-24.108,21.572,-43.334
C00524=1018.905,-34.581,-118.091,-24.109,21.571,-43.328
C00525=1018.906,-34.184,-118.123,-24.110,21.571,-43.321
C00526=1018.907,-33.786,-118.155,-24.111,21.570,-43.315
C00527=1018.907,-33.389,-118.186,-24.111,21.570,-43.310
C00528=1018.908,-32.991,-118.219,-24.112,21.570,-43.304
C00529=1018.909,-32.594,-118.251,-24.113,21.569,-43.299
C00530=1018.911,-32.196,-118.283,-24.114,21.568,-43.293
C00531=1018.911,-31.799,-118.315,-24.114,21.567,-43.287
C00532=1018.912,-31.401,-118.346,-24.115,21.568,-43.282
C00533=1018.913,-31.004,-118.379,-24.116,21.567,-43.277
C00534=1018.913,-30.607,-118.411,-24.117,21.566,-43.271
C00535=1018.914,-30.210,-118.443,-24.117,21.565,-43.265
C00536=1018.915,-29.812,-118.475,-24.118,21.565,-43.260
C00537=1018.915,-29.415,-118.507,-24.119,21.565,-43.255
C00538=1018.915,-29.017,-118.539,-24.120,21.564,-43.249
C00539=1018.916,-28.620,-118.572,-24.120,21.563,-43.243
C00540=1018.917,-28.222,-118.604,-24.121,21.562,-43.238
C00541=1018.918,-27.825,-118.636,-24.122,21.562,-43.232
C00542=1018.919,-27.427,-118.668,-24.123,21.562,-43.227
C00543=1018.920,-27.030,-118.701,-24.123,21.561,-43.221
C00544=1018.920,-26.632,-118.733,-24.124,21.560,-43.217
C00545=1018.920,-26.235,-118.765,-24.125,21.560,-43.212
C00546=1018.921,-25.837,-118.797,-24.125,21.559,-43.206
C00547=1018.921,-25.440,-118.830,-24.126,21.558,-43.201
C00548=1018.922,-25.043,-118.862,-24.127,21.558,-43.195
C00549=1018.923,-24.645,-118.894,-24.128,21.558,-43.190
C00550=1018.923,-24.248,-118.927,-24.128,21.557,-43.184
C00551=1018.924,-23.851,-118.959,-24.129,21.556,-43.178
C00552=1018.924,-23.453,-118.992,-24.130,21.556,-43.173
C00553=1018.924,-23.055,-119.023,-24.131,21.555,-43.168
C00554=1018.924,-22.658,-119.056,-24.131,21.555,-43.162
C00555=1018.925,-22.260,-119.088,-24.132,21.554,-43.156
C00556=1018.925,-21.862,-119.122,-24.133,21.554,-43.151
C00557=1018.926,-21.464,-119.154,-24.134,21.553,-43.146
C00558=1018.926,-21.067,-119.186,-24.134,21.552,-43.140
C00559=1018.926,-20.670,-119.219,-24.135,21.553,-43.135
C00560=1018.926,-20.272,-119.252,-24.136,21.552,-43.129
C00561=1018.927,-19.875,-119.284,-24.136,21.551,-43.123
C00562=1018.927,-19.464,-119.318,-24.138,21.551,-43.116
C00563=1018.927,-19.215,-119.339,-24.138,21.550,-43.113
C00564=1018.927,-18.926,-119.363,-24.139,21.550,-43.109
C00565=1018.928,-18.615,-119.388,-24.139,21.550,-43.107
C00566=1018.927,-18.304,-119.414,-24.139,21.549,-43.105
C00567=1018.928,-18.016,-119.437,-24.139,21.549,-43.101
C00568=1018.928,-17.768,-119.458,-24.140,21.548,-43.098
C00569=1018.929,-17.357,-119.492,-24.141,21.547,-43.090
C00570=1018.929,-16.960,-119.524,-24.142,21.548,-43.085
C00571=1018.929,-16.561,-119.556,-24.142,21.547,-43.079
C00572=1018.928,-16.163,-119.590,-24.143,21.546,-43.074
C00573=1018.929,-15.763,-119.623,-24.144,21.546,-43.068
C00574=1018.928,-15.362,-119.656,-24.145,21.545,-43.063
C00575=1018.929,-14.959,-119.689,-24.145,21.545,-43.057
C00576=1018.929,-14.554,-119.723,-24.146,21.544,-43.052
C00577=1018.929,-14.146,-119.757,-24.147,21.544,-43.046
C00578=1018.929,-13.734,-119.791,-24.148,21.543,-43.041
C00579=1018.929,-13.320,-119.825,-24.148,21.543,-43.035
C00580=1018.929,-12.902,-119.860,-24.149,21.542,-43.029
C00581=1018.929,-12.483,-119.895,-24.150,21.542,-43.024
C00582=1018.929,-12.272,-119.912,-24.150,21.541,-43.022
C00583=1018.929,-12.060,-119.930,-24.151,21.541,-43.019
C00584=1018.929,-11.848,-119.947,-24.151,21.540,-43.016
C00585=1018.928,-11.637,-119.965,-24.151,21.540,-43.013
C00586=1018.928,-11.424,-119.983,-24.152,21.540,-43.011
C00587=1018.929,-11.210,-120.001,-24.152,21.540,-43.007
C00588=1018.928,-10.996,-120.018,-24.152,21.539,-43.006
C00589=1018.929,-10.783,-120.036,-24.153,21.539,-43.002
C00590=1018.929,-10.567,-120.054,-24.153,21.539,-42.998
C00591=1018.929,-10.353,-120.072,-24.154,21.538,-42.996
C00592=1018.928,-10.137,-120.090,-24.154,21.539,-42.993
C00593=1018.928,-9.921,-120.108,-24.154,21.538,-42.991
C00594=1018.928,-9.706,-120.125,-24.155,21.538,-42.987
C00595=1018.928,-9.490,-120.143,-24.155,21.538,-42.985
C00596=1018.928,-9.273,-120.162,-24.156,21.537,-42.982
C00597=1018.928,-9.057,-120.180,-24.156,21.537,-42.980
C00598=1018.928,-8.841,-120.198,-24.156,21.536,-42.976
C00599=1018.928,-8.624,-120.216,-24.157,21.537,-42.973
C00600=1018.928,-8.407,-120.234,-24.157,21.536,-42.971
C00601=1018.927,-8.191,-120.252,-24.158,21.536,-42.967
C00602=1018.927,-7.974,-120.270,-24.158,21.536,-42.965
C00603=1018.928,-7.756,-120.288,-24.158,21.535,-42.961
C00604=1018.927,-7.538,-120.306,-24.159,21.535,-42.959
C00605=1018.927,-7.319,-120.325,-24.159,21.534,-42.956
C00606=1018.927,-7.099,-120.343,-24.160,21.535,-42.952
C00607=1018.927,-6.877,-120.362,-24.160,21.534,-42.950
C00608=1018.927,-6.655,-120.380,-24.160,21.534,-42.947
C00609=1018.926,-6.432,-120.399,-24.161,21.533,-42.944
C00610=1018.927,-6.208,-120.418,-24.161,21.533,-42.941
C00611=1018.926,-5.983,-120.436,-24.161,21.533,-42.939
C00612=1018.926,-5.760,-120.455,-24.162,21.533,-42.935
C00613=1018.925,-5.535,-120.475,-24.162,21.532,-42.934
C00614=1018.926,-5.312,-120.493,-24.163,21.532,-42.930
C00615=1018.925,-5.089,-120.512,-24.163,21.532,-42.927
C00616=1018.925,-4.868,-120.530,-24.163,21.532,-42.925
C00617=1018.924,-4.648,-120.549,-24.164,21.531,-42.921
C00618=1018.924,-4.429,-120.567,-24.164,21.531,-42.919
C00619=1018.924,-4.213,-120.585,-24.165,21.531,-42.915
C00620=1018.924,-3.997,-120.603,-24.165,21.530,-42.913
C00621=1018.924,-3.784,-120.621,-24.165,21.530,-42.910
C00622=1018.924,-3.571,-120.639,-24.166,21.530,-42.908
C00623=1018.923,-3.360,-120.657,-24.166,21.530,-42.904
C00624=1018.923,-2.939,-120.692,-24.167,21.529,-42.899
C00625=1018.922,-2.520,-120.728,-24.168,21.529,-42.893
C00626=1018.922,-2.102,-120.763,-24.169,21.529,-42.888
C00627=1018.922,-1.687,-120.797,-24.169,21.528,-42.882
C00628=1018.921,-1.274,-120.832,-24.170,21.527,-42.877
C00629=1018.920,-0.865,-120.867,-24.171,21.527,-42.872
C00630=1018.920,-0.456,-120.901,-24.171,21.526,-42.867
C00631=1018.920,-0.051,-120.936,-24.172,21.525,-42.862
C00632=1018.919,0.352,-120.970,-24.173,21.525,-42.857
C00633=1018.918,0.754,-121.004,-24.173,21.525,-42.851
C00634=1018.918,1.155,-121.038,-24.174,21.525,-42.846
C00635=1018.917,1.552,-121.071,-24.175,21.523,-42.841
C00636=1018.917,1.951,-121.105,-24.175,21.524,-42.836
C00637=1018.916,2.337,-121.138,-24.176,21.523,-42.833
C00638=1018.915,2.689,-121.168,-24.177,21.522,-42.827
C00639=1018.915,3.012,-121.195,-24.177,21.522,-42.823
C00640=1018.915,3.326,-121.221,-24.178,21.521,-42.817
C00641=1018.914,3.654,-121.249,-24.179,21.521,-42.812
C00642=1018.913,4.013,-121.280,-24.179,21.521,-42.809
C00643=1018.912,4.402,-121.313,-24.180,21.520,-42.805
C00644=1018.911,4.798,-121.347,-24.180,21.519,-42.799
C00645=1018.910,5.194,-121.380,-24.181,21.520,-42.794
C00646=1018.910,5.589,-121.413,-24.182,21.519,-42.790
C00647=1018.909,5.983,-121.448,-24.182,21.518,-42.785
C00648=1018.909,6.376,-121.481,-24.183,21.519,-42.779
C00649=1018.907,6.769,-121.515,-24.184,21.517,-42.775
C00650=1018.907,7.162,-121.548,-24.185,21.517,-42.770
C00651=1018.906,7.552,-121.582,-24.185,21.517,-42.764
C00652=1018.905,7.940,-121.614,-24.186,21.516,-42.761
C00653=1018.904,8.324,-121.647,-24.187,21.516,-42.755
C00654=1018.903,8.705,-121.680,-24.187,21.515,-42.751
C00655=1018.902,9.083,-121.712,-24.188,21.515,-42.746
C00656=1018.901,9.459,-121.744,-24.189,21.514,-42.740
C00657=1018.900,9.835,-121.776,-24.189,21.514,-42.737
C00658=1018.899,10.211,-121.809,-24.190,21.513,-42.731
C00659=1018.899,10.590,-121.841,-24.191,21.513,-42.726
C00660=1018.898,10.970,-121.874,-24.191,21.513,-42.722
C00661=1018.896,11.354,-121.907,-24.192,21.512,-42.716
C00662=1018.895,11.739,-121.940,-24.192,21.511,-42.713
C00663=1018.895,12.126,-121.973,-24.193,21.512,-42.707
C00664=1018.893,12.512,-122.006,-24.193,21.510,-42.703
C00665=1018.893,12.898,-122.039,-24.194,21.510,-42.698
C00666=1018.892,13.285,-122.073,-24.195,21.511,-42.693
C00667=1018.890,13.672,-122.106,-24.196,21.509,-42.689
C00668=1018.889,14.059,-122.140,-24.196,21.509,-42.683
C00669=1018.888,14.447,-122.173,-24.197,21.509,-42.680
C00670=1018.887,14.835,-122.206,-24.198,21.508,-42.674
C00671=1018.886,15.224,-122.240,-24.198,21.508,-42.670
C00672=1018.885,15.614,-122.273,-24.199,21.507,-42.665
C00673=1018.883,16.004,-122.307,-24.200,21.507,-42.659
C00674=1018.882,16.395,-122.341,-24.200,21.506,-42.656
C00675=1018.881,16.787,-122.375,-24.201,21.506,-42.650
C00676=1018.880,17.179,-122.409,-24.201,21.505,-42.646
C00677=1018.879,17.572,-122.442,-24.202,21.505,-42.641
C00678=1018.877,17.967,-122.476,-24.203,21.505,-42.635
C00679=1018.876,18.362,-122.511,-24.203,21.504,-42.632
C00680=1018.875,18.758,-122.545,-24.204,21.503,-42.626
C00681=1018.873,19.154,-122.580,-24.205,21.503,-42.622
C00682=1018.872,19.552,-122.614,-24.205,21.503,-42.617
C00683=1018.871,19.763,-122.632,-24.206,21.503,-42.613
C00684=1018.870,19.999,-122.652,-24.206,21.502,-42.610
C00685=1018.870,20.264,-122.675,-24.207,21.503,-42.606
C00686=1018.868,20.552,-122.700,-24.207,21.501,-42.604
C00687=1018.867,20.848,-122.726,-24.207,21.501,-42.602
C00688=1018.867,21.140,-122.752,-24.208,21.502,-42.599
C00689=1018.866,21.412,-122.775,-24.208,21.501,-42.597
C00690=1018.865,21.657,-122.797,-24.209,21.501,-42.593
C00691=1018.863,22.070,-122.833,-24.210,21.501,-42.586
C00692=1018.862,22.445,-122.865,-24.210,21.500,-42.584
C00693=1018.860,22.767,-122.893,-24.211,21.500,-42.580
C00694=1018.860,23.033,-122.916,-24.211,21.500,-42.577
C00695=1018.859,23.265,-122.936,-24.211,21.499,-42.573
C00696=1018.858,23.499,-122.957,-24.212,21.498,-42.567
C00697=1018.858,23.771,-122.981,-24.213,21.498,-42.564
C00698=1018.855,24.101,-123.010,-24.213,21.498,-42.562
C00699=1018.854,24.485,-123.043,-24.213,21.497,-42.558
C00700=1018.853,24.884,-123.078,-24.214,21.497,-42.553
C00701=1018.851,25.283,-123.113,-24.215,21.497,-42.549
C00702=1018.849,25.683,-123.147,-24.215,21.496,-42.543
C00703=1018.848,26.082,-123.182,-24.216,21.496,-42.540
C00704=1018.846,26.482,-123.217,-24.217,21.496,-42.534
C00705=1018.845,26.881,-123.252,-24.218,21.495,-42.529
C00706=1018.843,27.280,-123.287,-24.218,21.494,-42.525
C00707=1018.841,27.679,-123.322,-24.219,21.495,-42.520
C00708=1018.840,28.078,-123.357,-24.219,21.493,-42.516
C00709=1018.838,28.478,-123.393,-24.220,21.493,-42.510
C00710=1018.837,28.878,-123.428,-24.221,21.493,-42.507
C00711=1018.835,29.278,-123.462,-24.221,21.492,-42.501
C00712=1018.833,29.677,-123.497,-24.222,21.492,-42.497
C00713=1018.831,30.076,-123.533,-24.223,21.492,-42.492
C00714=1018.829,30.476,-123.567,-24.223,21.491,-42.488
C00715=1018.828,30.876,-123.603,-24.224,21.491,-42.483
C00716=1018.826,31.275,-123.638,-24.224,21.490,-42.479
C00717=1018.824,31.674,-123.673,-24.225,21.490,-42.474
C00718=1018.822,32.075,-123.708,-24.226,21.489,-42.469
C00719=1018.820,32.474,-123.743,-24.226,21.489,-42.464
C00720=1018.818,32.874,-123.779,-24.227,21.489,-42.461
C00721=1018.817,33.273,-123.814,-24.228,21.489,-42.455
C00722=1018.814,33.673,-123.849,-24.228,21.487,-42.451
C00723=1018.813,34.073,-123.885,-24.229,21.488,-42.446
C00724=1018.811,34.473,-123.919,-24.229,21.487,-42.442
C00725=1018.808,34.872,-123.955,-24.230,21.486,-42.437
C00726=1018.807,35.272,-123.990,-24.231,21.486,-42.433
C00727=1018.805,35.672,-124.026,-24.231,21.486,-42.428
C00728=1018.803,36.071,-124.061,-24.232,21.486,-42.424
C00729=1018.801,36.471,-124.096,-24.233,21.485,-42.418
C00730=1018.799,36.871,-124.131,-24.233,21.484,-42.414
C00731=1018.797,37.271,-124.167,-24.234,21.485,-42.409
C00732=1018.795,37.670,-124.202,-24.235,21.484,-42.405
C00733=1018.793,38.071,-124.238,-24.235,21.483,-42.400
C00734=1018.790,38.470,-124.274,-24.236,21.483,-42.396
C00735=1018.789,38.871,-124.308,-24.237,21.483,-42.391
C00736=1018.787,39.270,-124.344,-24.237,21.483,-42.387
C00737=1018.785,39.670,-124.379,-24.238,21.482,-42.383
C00738=1018.783,40.070,-124.415,-24.238,21.481,-42.378
C00739=1018.780,40.470,-124.451,-24.239,21.481,-42.374
C00740=1018.778,40.869,-124.486,-24.240,21.481,-42.369
C00741=1018.776,41.270,-124.522,-24.240,21.481,-42.365
C00742=1018.773,41.670,-124.558,-24.241,21.480,-42.359
C00743=1018.771,42.070,-124.594,-24.241,21.479,-42.356
C00744=1018.769,42.470,-124.629,-24.242,21.479,-42.352
C00745=1018.767,42.870,-124.665,-24.243,21.479,-42.347
C00746=1018.765,43.270,-124.700,-24.243,21.479,-42.343
C00747=1018.762,43.670,-124.735,-24.244,21.479,-42.338
C00748=1018.760,44.070,-124.772,-24.244,21.477,-42.333
C00749=1018.758,44.470,-124.807,-24.245,21.477,-42.330
C00750=1018.756,44.870,-124.843,-24.246,21.477,-42.325
C00751=1018.753,45.269,-124.879,-24.246,21.477,-42.321
C00752=1018.751,45.671,-124.915,-24.247,21.477,-42.316
C00753=1018.748,46.070,-124.950,-24.247,21.475,-42.311
C00754=1018.747,46.470,-124.986,-24.248,21.475,-42.308
C00755=1018.744,46.870,-125.022,-24.249,21.475,-42.302
C00756=1018.742,47.271,-125.058,-24.249,21.475,-42.299
C00757=1018.738,47.671,-125.093,-24.250,21.474,-42.295
C00758=1018.736,48.071,-125.129,-24.251,21.474,-42.290
C00759=1018.734,48.471,-125.165,-24.251,21.474,-42.286
C00760=1018.731,48.871,-125.201,-24.251,21.472,-42.282
C00761=1018.729,49.271,-125.237,-24.252,21.473,-42.277
C00762=1018.727,49.671,-125.273,-24.253,21.472,-42.273
C00763=1018.724,50.072,-125.309,-24.254,21.472,-42.268
C00764=1018.721,50.471,-125.344,-24.254,21.472,-42.264
C00765=1018.719,50.872,-125.381,-24.255,21.471,-42.260
C00766=1018.716,51.272,-125.417,-24.255,21.471,-42.255
C00767=1018.714,51.672,-125.453,-24.256,21.471,-42.251
C00768=1018.711,52.072,-125.489,-24.256,21.470,-42.247
C00769=1018.709,52.473,-125.525,-24.257,21.469,-42.243
C00770=1018.706,52.872,-125.561,-24.258,21.469,-42.238
C00771=1018.704,53.273,-125.597,-24.258,21.469,-42.234
C00772=1018.700,53.673,-125.633,-24.259,21.468,-42.230
C00773=1018.697,54.073,-125.669,-24.259,21.468,-42.225
C00774=1018.695,54.473,-125.705,-24.260,21.468,-42.221
C00775=1018.693,54.873,-125.741,-24.260,21.468,-42.218
C00776=1018.690,55.274,-125.777,-24.261,21.468,-42.212
C00777=1018.687,55.673,-125.813,-24.262,21.467,-42.209
C00778=1018.685,56.074,-125.850,-24.262,21.467,-42.205
C00779=1018.682,56.474,-125.886,-24.263,21.465,-42.201
C00780=1018.679,56.875,-125.922,-24.264,21.466,-42.196
C00781=1018.676,57.275,-125.958,-24.264,21.465,-42.192
C00782=1018.673,57.675,-125.994,-24.264,21.465,-42.188
C00783=1018.670,58.075,-126.031,-24.265,21.465,-42.183
C00784=1018.667,58.475,-126.067,-24.266,21.464,-42.179
C00785=1018.665,58.876,-126.103,-24.266,21.464,-42.175
C00786=1018.662,59.276,-126.139,-24.267,21.463,-42.172
C00787=1018.659,59.676,-126.176,-24.268,21.464,-42.166
C00788=1018.656,60.076,-126.212,-24.268,21.463,-42.163
C00789=1018.653,60.476,-126.248,-24.269,21.463,-42.159
C00790=1018.651,60.876,-126.285,-24.269,21.462,-42.155
C00791=1018.647,61.276,-126.321,-24.270,21.462,-42.150
C00792=1018.644,61.677,-126.358,-24.270,21.462,-42.146
C00793=1018.641,62.077,-126.394,-24.271,21.461,-42.142
C00794=1018.638,62.477,-126.430,-24.271,21.461,-42.139
C00795=1018.635,62.896,-126.468,-24.272,21.460,-42.133
C00796=1018.633,63.150,-126.492,-24.272,21.460,-42.131
C00797=1018.631,63.417,-126.516,-24.273,21.460,-42.129
C00798=1018.629,63.667,-126.539,-24.273,21.459,-42.127
C00799=1018.628,63.885,-126.558,-24.274,21.460,-42.124
C00800=1018.626,64.092,-126.577,-24.274,21.460,-42.122
C00801=1018.625,64.310,-126.597,-24.274,21.459,-42.120
C00802=1018.623,64.538,-126.618,-24.274,21.459,-42.116
C00803=1018.621,64.775,-126.639,-24.275,21.459,-42.115
C00804=1018.619,65.011,-126.660,-24.275,21.458,-42.113
C00805=1018.617,65.241,-126.682,-24.275,21.458,-42.111
C00806=1018.615,65.462,-126.702,-24.276,21.459,-42.108
C00807=1018.614,65.675,-126.721,-24.276,21.458,-42.106
C00808=1018.611,66.083,-126.759,-24.277,21.458,-42.102
C00809=1018.607,66.481,-126.795,-24.277,21.457,-42.098
C00810=1018.605,66.881,-126.831,-24.278,21.457,-42.094
C00811=1018.601,67.284,-126.868,-24.278,21.457,-42.089
C00812=1018.598,67.687,-126.905,-24.279,21.457,-42.085
C00813=1018.595,68.092,-126.941,-24.279,21.456,-42.082
C00814=1018.592,68.498,-126.979,-24.280,21.456,-42.078
C00815=1018.589,68.906,-127.016,-24.280,21.455,-42.074
C00816=1018.585,69.314,-127.053,-24.281,21.455,-42.069
C00817=1018.582,69.724,-127.091,-24.282,21.455,-42.065
C00818=1018.578,70.135,-127.129,-24.282,21.454,-42.061
C00819=1018.575,70.547,-127.167,-24.283,21.454,-42.058
C00820=1018.572,70.958,-127.203,-24.283,21.453,-42.054
C00821=1018.568,71.369,-127.241,-24.284,21.454,-42.049
C00822=1018.564,71.780,-127.279,-24.285,21.453,-42.045
C00823=1018.561,72.192,-127.317,-24.285,21.453,-42.041
C00824=1018.557,72.606,-127.355,-24.285,21.452,-42.037
C00825=1018.555,73.021,-127.393,-24.286,21.452,-42.034
C00826=1018.550,73.439,-127.432,-24.287,21.452,-42.028
C00827=1018.547,73.859,-127.470,-24.287,21.452,-42.025
C00828=1018.545,74.071,-127.489,-24.288,21.451,-42.023
C00829=1018.544,74.283,-127.509,-24.288,21.451,-42.021
C00830=1018.542,74.495,-127.528,-24.288,21.451,-42.019
C00831=1018.540,74.708,-127.549,-24.288,21.451,-42.017
C00832=1018.538,74.922,-127.568,-24.289,21.450,-42.015
C00833=1018.536,75.136,-127.587,-24.289,21.451,-42.012
C00834=1018.534,75.349,-127.607,-24.289,21.451,-42.010
C00835=1018.532,75.561,-127.626,-24.290,21.450,-42.008
C00836=1018.528,75.981,-127.665,-24.290,21.450,-42.004
C00837=1018.525,76.393,-127.703,-24.291,21.449,-42.001
C00838=1018.522,76.795,-127.740,-24.291,21.449,-41.997
C00839=1018.518,77.190,-127.776,-24.292,21.449,-41.994
C00840=1018.514,77.578,-127.812,-24.292,21.448,-41.989
C00841=1018.511,77.964,-127.848,-24.293,21.447,-41.986
C00842=1018.508,78.351,-127.883,-24.293,21.448,-41.980
C00843=1018.504,78.741,-127.919,-24.294,21.447,-41.977
C00844=1018.501,79.139,-127.955,-24.294,21.447,-41.973
C00845=1018.497,79.543,-127.993,-24.295,21.447,-41.970
C00846=1018.493,79.958,-128.032,-24.296,21.447,-41.966
C00847=1018.491,80.169,-128.051,-24.296,21.446,-41.964
C00848=1018.489,80.380,-128.071,-24.296,21.446,-41.962
C00849=1018.488,80.593,-128.090,-24.296,21.446,-41.960
C00850=1018.486,80.805,-128.110,-24.297,21.446,-41.958
C00851=1018.483,81.019,-128.129,-24.297,21.445,-41.956
C00852=1018.481,81.232,-128.149,-24.297,21.445,-41.955
C00853=1018.480,81.444,-128.169,-24.297,21.445,-41.953
C00854=1018.477,81.657,-128.189,-24.298,21.445,-41.951
C00855=1018.475,81.869,-128.208,-24.298,21.445,-41.949
C00856=1018.473,82.080,-128.228,-24.298,21.444,-41.947
C00857=1018.472,82.292,-128.247,-24.299,21.445,-41.944
C00858=1018.470,82.503,-128.266,-24.299,21.444,-41.942
C00859=1018.467,82.714,-128.286,-24.299,21.444,-41.940
C00860=1018.466,82.924,-128.305,-24.299,21.444,-41.938
C00861=1018.462,83.345,-128.344,-24.300,21.444,-41.935
C00862=1018.458,83.763,-128.383,-24.300,21.444,-41.931
C00863=1018.454,84.181,-128.422,-24.301,21.443,-41.927
C00864=1018.450,84.596,-128.460,-24.301,21.443,-41.923
C00865=1018.446,85.011,-128.499,-24.302,21.443,-41.920
C00866=1018.442,85.423,-128.538,-24.302,21.442,-41.916
C00867=1018.438,85.834,-128.575,-24.303,21.442,-41.912
C00868=1018.434,86.243,-128.613,-24.303,21.441,-41.908
C00869=1018.429,86.650,-128.651,-24.304,21.442,-41.905
C00870=1018.426,87.055,-128.689,-24.304,21.441,-41.901
C00871=1018.422,87.459,-128.725,-24.305,21.441,-41.898
C00872=1018.419,87.855,-128.763,-24.305,21.440,-41.894
C00873=1018.415,88.243,-128.799,-24.306,21.440,-41.890
C00874=1018.410,88.626,-128.834,-24.307,21.440,-41.887
C00875=1018.407,89.009,-128.870,-24.307,21.440,-41.883
C00876=1018.403,89.396,-128.906,-24.308,21.439,-41.879
C00877=1018.399,89.789,-128.942,-24.308,21.439,-41.875
C00878=1018.395,90.187,-128.979,-24.309,21.439,-41.872
C00879=1018.390,90.586,-129.017,-24.309,21.439,-41.868
C00880=1018.387,90.986,-129.054,-24.310,21.438,-41.865
C00881=1018.383,91.385,-129.091,-24.310,21.438,-41.861
C00882=1018.379,91.783,-129.128,-24.311,21.438,-41.857
C00883=1018.374,92.183,-129.166,-24.311,21.438,-41.854
C00884=1018.370,92.582,-129.203,-24.312,21.437,-41.850
C00885=1018.366,92.982,-129.239,-24.312,21.437,-41.846
C00886=1018.362,93.380,-129.277,-24.312,21.437,-41.844
C00887=1018.358,93.779,-129.314,-24.313,21.436,-41.841
C00888=1018.354,94.178,-129.351,-24.313,21.436,-41.837
C00889=1018.349,94.578,-129.389,-24.314,21.435,-41.833
C00890=1018.345,94.977,-129.426,-24.315,21.436,-41.830
C00891=1018.341,95.376,-129.463,-24.315,21.435,-41.826
C00892=1018.337,95.774,-129.500,-24.316,21.435,-41.822
C00893=1018.332,96.173,-129.538,-24.316,21.435,-41.819
C00894=1018.328,96.572,-129.575,-24.317,21.435,-41.815
C00895=1018.324,96.971,-129.612,-24.317,21.434,-41.811
C00896=1018.319,97.370,-129.649,-24.318,21.434,-41.808
C00897=1018.315,97.769,-129.686,-24.318,21.433,-41.806
C00898=1018.311,98.167,-129.724,-24.318,21.433,-41.802
C00899=1018.307,98.566,-129.762,-24.319,21.432,-41.798
C00900=1018.303,98.965,-129.799,-24.319,21.433,-41.795
C00901=1018.298,99.364,-129.836,-24.320,21.432,-41.791
C00902=1018.294,99.763,-129.874,-24.320,21.432,-41.787
C00903=1018.289,100.162,-129.911,-24.321,21.432,-41.784
C00904=1018.284,100.560,-129.948,-24.322,21.432,-41.780
C00905=1018.280,100.959,-129.985,-24.322,21.431,-41.778
C00906=1018.276,101.358,-130.022,-24.322,21.431,-41.775
C00907=1018.271,101.757,-130.060,-24.323,21.431,-41.771
C00908=1018.267,102.155,-130.098,-24.323,21.430,-41.767
C00909=1018.262,102.555,-130.135,-24.324,21.430,-41.763
C00910=1018.258,102.953,-130.172,-24.324,21.430,-41.760
C00911=1018.253,103.352,-130.210,-24.325,21.430,-41.756
C00912=1018.249,103.750,-130.247,-24.325,21.430,-41.754
C00913=1018.244,104.149,-130.285,-24.326,21.429,-41.751
C00914=1018.240,104.548,-130.322,-24.326,21.429,-41.747
C00915=1018.235,104.946,-130.359,-24.327,21.429,-41.743
C00916=1018.231,105.345,-130.396,-24.327,21.429,-41.740
C00917=1018.226,105.744,-130.435,-24.328,21.428,-41.736
C00918=1018.221,106.142,-130.472,-24.328,21.428,-41.734
C00919=1018.217,106.541,-130.509,-24.328,21.427,-41.730
C00920=1018.212,106.940,-130.547,-24.329,21.427,-41.727
C00921=1018.207,107.338,-130.584,-24.330,21.427,-41.723
C00922=1018.203,107.737,-130.622,-24.330,21.427,-41.719
C00923=1018.198,108.136,-130.660,-24.330,21.426,-41.717
C00924=1018.193,108.534,-130.696,-24.331,21.426,-41.714
C00925=1018.188,108.933,-130.735,-24.331,21.426,-41.710
C00926=1018.184,109.332,-130.772,-24.332,21.426,-41.707
C00927=1018.179,109.730,-130.809,-24.332,21.426,-41.703
C00928=1018.174,110.128,-130.847,-24.333,21.425,-41.701
C00929=1018.169,110.527,-130.885,-24.333,21.425,-41.697
C00930=1018.164,110.926,-130.922,-24.334,21.425,-41.694
C00931=1018.160,111.323,-130.960,-24.334,21.425,-41.690
C00932=1018.155,111.722,-130.997,-24.334,21.424,-41.688
C00933=1018.150,112.122,-131.035,-24.335,21.423,-41.684
C00934=1018.145,112.520,-131.072,-24.335,21.424,-41.681
C00935=1018.140,112.919,-131.111,-24.336,21.423,-41.677
C00936=1018.135,113.317,-131.147,-24.336,21.423,-41.675
C00937=1018.131,113.716,-131.185,-24.337,21.423,-41.671
C00938=1018.125,114.114,-131.223,-24.337,21.422,-41.668
C00939=1018.121,114.513,-131.261,-24.338,21.423,-41.664
C00940=1018.115,114.911,-131.298,-24.338,21.422,-41.662
C00941=1018.111,115.310,-131.336,-24.339,21.422,-41.659
C00942=1018.105,115.708,-131.374,-24.339,21.422,-41.655
C00943=1018.100,116.106,-131.412,-24.340,21.422,-41.652
C00944=1018.095,116.505,-131.449,-24.340,21.421,-41.649
C00945=1018.090,116.939,-131.490,-24.340,21.420,-41.646
C00946=1018.085,117.302,-131.525,-24.341,21.421,-41.642
C00947=1018.080,117.700,-131.562,-24.341,21.420,-41.638
C00948=1018.075,118.100,-131.600,-24.342,21.420,-41.637
C00949=1018.070,118.497,-131.638,-24.342,21.420,-41.633
C00950=1018.064,118.896,-131.675,-24.343,21.420,-41.629
C00951=1018.060,119.295,-131.713,-24.343,21.420,-41.626
C00952=1018.054,119.693,-131.751,-24.343,21.419,-41.624
C00953=1018.049,120.091,-131.788,-24.344,21.419,-41.620
C00954=1018.045,120.490,-131.827,-24.345,21.419,-41.617
C00955=1018.040,120.889,-131.864,-24.345,21.418,-41.614
C00956=1018.035,121.287,-131.902,-24.345,21.418,-41.611
C00957=1018.030,121.686,-131.940,-24.346,21.418,-41.607
C00958=1018.024,122.085,-131.979,-24.346,21.417,-41.605
C00959=1018.019,122.482,-132.017,-24.347,21.418,-41.602
C00960=1018.015,122.882,-132.055,-24.347,21.417,-41.598
C00961=1018.010,123.280,-132.093,-24.348,21.418,-41.595
C00962=1018.005,123.678,-132.130,-24.348,21.416,-41.592
C00963=1018.000,124.077,-132.169,-24.348,21.417,-41.589
C00964=1017.995,124.475,-132.207,-24.349,21.416,-41.585
C00965=1017.990,124.874,-132.244,-24.349,21.416,-41.583
C00966=1017.985,125.273,-132.283,-24.350,21.416,-41.580
C00967=1017.980,125.671,-132.321,-24.350,21.416,-41.576
C00968=1017.975,126.070,-132.359,-24.350,21.415,-41.574
C00969=1017.970,126.468,-132.397,-24.351,21.415,-41.571
C00970=1017.964,126.867,-132.435,-24.351,21.415,-41.567
C00971=1017.960,127.265,-132.473,-24.352,21.415,-41.565
C00972=1017.955,127.664,-132.512,-24.352,21.414,-41.561
C00973=1017.949,128.063,-132.550,-24.353,21.415,-41.558
C00974=1017.944,128.461,-132.588,-24.353,21.414,-41.555
C00975=1017.939,128.860,-132.625,-24.354,21.414,-41.552
C00976=1017.934,129.258,-132.664,-24.354,21.413,-41.550
C00977=1017.929,129.658,-132.702,-24.354,21.413,-41.547
C00978=1017.923,130.056,-132.741,-24.355,21.413,-41.543
C00979=1017.918,130.454,-132.779,-24.355,21.413,-41.541
C00980=1017.913,130.853,-132.816,-24.356,21.413,-41.538
C00981=1017.908,131.252,-132.855,-24.356,21.413,-41.534
C00982=1017.903,131.651,-132.893,-24.356,21.412,-41.532
C00983=1017.897,132.049,-132.932,-24.357,21.412,-41.528
C00984=1017.891,132.448,-132.970,-24.357,21.412,-41.525
C00985=1017.886,132.846,-133.008,-24.358,21.411,-41.523
C00986=1017.881,133.245,-133.047,-24.358,21.412,-41.519
C00987=1017.876,133.644,-133.084,-24.358,21.411,-41.517
C00988=1017.870,134.042,-133.123,-24.359,21.411,-41.514
C00989=1017.866,134.441,-133.161,-24.359,21.411,-41.510
C00990=1017.860,134.839,-133.199,-24.360,21.410,-41.508
C00991=1017.854,135.239,-133.238,-24.360,21.411,-41.505
C00992=1017.849,135.634,-133.276,-24.360,21.410,-41.502
C00993=1017.844,136.005,-133.311,-24.361,21.409,-41.500
C00994=1017.839,136.345,-133.343,-24.361,21.410,-41.497
C00995=1017.835,136.662,-133.375,-24.361,21.409,-41.495
C00996=1017.831,136.979,-133.404,-24.362,21.409,-41.491
C00997=1017.826,137.315,-133.437,-24.363,21.410,-41.488
C00998=1017.820,137.685,-133.473,-24.363,21.408,-41.486
C00999=1017.815,138.087,-133.511,-24.363,21.408,-41.484
C01000=1017.812,138.293,-133.531,-24.363,21.408,-41.482
C01001=1017.809,138.509,-133.552,-24.364,21.408,-41.480
C01002=1017.805,138.747,-133.574,-24.364,21.408,-41.478
C01003=1017.802,139.006,-133.599,-24.364,21.407,-41.476
C01004=1017.798,139.284,-133.627,-24.364,21.408,-41.475
C01005=1017.794,139.572,-133.654,-24.365,21.408,-41.473
C01006=1017.790,139.859,-133.682,-24.365,21.408,-41.471
C01007=1017.786,140.137,-133.709,-24.365,21.408,-41.470
C01008=1017.782,140.395,-133.733,-24.366,21.408,-41.468
C01009=1017.779,140.631,-133.756,-24.366,21.408,-41.466
C01010=1017.774,141.049,-133.796,-24.366,21.407,-41.462
C01011=1017.768,141.452,-133.835,-24.366,21.406,-41.460
C01012=1017.762,141.859,-133.874,-24.367,21.407,-41.457
C01013=1017.756,142.265,-133.914,-24.368,21.406,-41.453
C01014=1017.750,142.672,-133.952,-24.368,21.406,-41.451
C01015=1017.745,143.080,-133.992,-24.368,21.406,-41.448
C01016=1017.739,143.488,-134.031,-24.369,21.405,-41.445
C01017=1017.733,143.898,-134.070,-24.369,21.406,-41.442
C01018=1017.727,144.309,-134.110,-24.370,21.405,-41.438
C01019=1017.721,144.719,-134.149,-24.370,21.405,-41.436
C01020=1017.715,145.131,-134.189,-24.370,21.405,-41.432
C01021=1017.708,145.543,-134.229,-24.371,21.404,-41.431
C01022=1017.703,145.955,-134.269,-24.371,21.405,-41.427
C01023=1017.697,146.368,-134.308,-24.372,21.404,-41.424
C01024=1017.691,146.781,-134.349,-24.372,21.404,-41.422
C01025=1017.684,147.195,-134.388,-24.372,21.404,-41.418
C01026=1017.678,147.608,-134.428,-24.373,21.403,-41.416
C01027=1017.672,148.022,-134.468,-24.373,21.403,-41.412
C01028=1017.666,148.437,-134.508,-24.374,21.403,-41.409
C01029=1017.660,148.850,-134.548,-24.374,21.403,-41.407
C01030=1017.654,149.264,-134.588,-24.375,21.403,-41.403
C01031=1017.647,149.678,-134.628,-24.375,21.402,-41.401
C01032=1017.641,150.093,-134.668,-24.375,21.402,-41.398
C01033=1017.635,150.507,-134.708,-24.376,21.402,-41.394
C01034=1017.629,150.920,-134.747,-24.376,21.401,-41.392
C01035=1017.622,151.334,-134.787,-24.377,21.402,-41.389
C01036=1017.616,151.747,-134.828,-24.377,21.402,-41.387
C01037=1017.610,152.160,-134.867,-24.377,21.401,-41.383
C01038=1017.603,152.573,-134.908,-24.378,21.401,-41.381
C01039=1017.597,152.985,-134.947,-24.378,21.400,-41.377
C01040=1017.591,153.397,-134.988,-24.378,21.400,-41.375
C01041=1017.584,153.808,-135.027,-24.379,21.401,-41.372
C01042=1017.578,154.219,-135.067,-24.380,21.400,-41.368
C01043=1017.571,154.629,-135.106,-24.380,21.400,-41.366
C01044=1017.566,155.038,-135.146,-24.380,21.400,-41.363
C01045=1017.559,155.446,-135.185,-24.381,21.399,-41.361
C01046=1017.553,155.854,-135.225,-24.381,21.400,-41.358
C01047=1017.546,156.261,-135.264,-24.381,21.399,-41.355
C01048=1017.540,156.667,-135.304,-24.382,21.399,-41.352
C01049=1017.533,157.072,-135.342,-24.382,21.399,-41.350
C01050=1017.527,157.476,-135.382,-24.383,21.398,-41.346
C01051=1017.520,157.879,-135.421,-24.383,21.398,-41.344
C01052=1017.514,158.282,-135.460,-24.383,21.399,-41.341
C01053=1017.508,158.684,-135.499,-24.384,21.397,-41.339
C01054=1017.501,159.085,-135.538,-24.384,21.398,-41.335
C01055=1017.494,159.486,-135.576,-24.384,21.398,-41.333
C01056=1017.491,159.886,-135.617,-24.385,21.397,-41.330
C01057=1017.490,160.283,-135.659,-24.385,21.397,-41.328
C01058=1017.489,160.688,-135.701,-24.386,21.397,-41.325
C01059=1017.488,160.902,-135.724,-24.386,21.397,-41.324
C01060=1017.487,161.125,-135.747,-24.386,21.396,-41.322
C01061=1017.486,161.363,-135.772,-24.386,21.396,-41.320
C01062=1017.485,161.615,-135.798,-24.387,21.397,-41.319
C01063=1017.484,161.877,-135.826,-24.387,21.397,-41.317
C01064=1017.484,162.146,-135.854,-24.387,21.396,-41.315
C01065=1017.482,162.418,-135.883,-24.387,21.396,-41.313
C01066=1017.482,162.686,-135.911,-24.388,21.396,-41.311
C01067=1017.481,162.950,-135.938,-24.388,21.396,-41.309
C01068=1017.480,163.204,-135.965,-24.388,21.395,-41.308
C01069=1017.479,163.439,-135.990,-24.388,21.396,-41.306
C01070=1017.478,163.850,-136.033,-24.389,21.395,-41.304
C01071=1017.477,164.040,-136.053,-24.389,21.395,-41.302
C01072=1017.476,164.426,-136.093,-24.389,21.395,-41.300
C01073=1017.474,164.826,-136.136,-24.390,21.395,-41.297
C01074=1017.473,165.227,-136.178,-24.390,21.395,-41.295
C01075=1017.472,165.628,-136.221,-24.390,21.394,-41.291
C01076=1017.470,166.028,-136.262,-24.391,21.394,-41.289
C01077=1017.469,166.428,-136.305,-24.391,21.395,-41.286
C01078=1017.467,166.828,-136.346,-24.391,21.393,-41.284
C01079=1017.466,167.229,-136.389,-24.392,21.394,-41.280
C01080=1017.465,167.630,-136.431,-24.392,21.394,-41.278
C01081=1017.464,168.030,-136.474,-24.393,21.394,-41.275
C01082=1017.463,168.430,-136.516,-24.393,21.393,-41.273
C01083=1017.461,168.831,-136.558,-24.393,21.393,-41.271
C01084=1017.460,169.231,-136.601,-24.394,21.393,-41.267
C01085=1017.459,169.632,-136.642,-24.394,21.392,-41.265
C01086=1017.457,170.032,-136.685,-24.395,21.392,-41.262
C01087=1017.456,170.433,-136.727,-24.395,21.392,-41.260
C01088=1017.454,170.833,-136.770,-24.395,21.392,-41.256
C01089=1017.453,171.234,-136.812,-24.396,21.392,-41.254
C01090=1017.452,171.634,-136.854,-24.396,21.392,-41.251
C01091=1017.451,172.035,-136.897,-24.396,21.392,-41.249
C01092=1017.449,172.435,-136.940,-24.397,21.391,-41.247
C01093=1017.449,172.836,-136.982,-24.397,21.391,-41.243
C01094=1017.447,173.237,-137.025,-24.397,21.391,-41.242
C01095=1017.446,173.637,-137.068,-24.398,21.390,-41.238
C01096=1017.444,174.038,-137.110,-24.398,21.390,-41.236
C01097=1017.444,174.439,-137.152,-24.399,21.391,-41.233
C01098=1017.442,174.839,-137.195,-24.399,21.390,-41.231
C01099=1017.441,175.240,-137.237,-24.400,21.390,-41.227
C01100=1017.439,175.641,-137.280,-24.400,21.390,-41.225
C01101=1017.439,176.042,-137.323,-24.400,21.390,-41.223
C01102=1017.438,176.443,-137.365,-24.401,21.389,-41.219
C01103=1017.436,176.843,-137.408,-24.401,21.389,-41.218
C01104=1017.435,177.244,-137.451,-24.401,21.389,-41.214
C01105=1017.434,177.644,-137.494,-24.402,21.389,-41.212
C01106=1017.433,178.046,-137.536,-24.402,21.389,-41.209
C01107=1017.432,178.446,-137.579,-24.402,21.388,-41.207
C01108=1017.431,178.847,-137.622,-24.403,21.388,-41.205
C01109=1017.429,179.247,-137.665,-24.403,21.388,-41.201
C01110=1017.428,179.649,-137.708,-24.403,21.388,-41.199
C01111=1017.427,180.050,-137.750,-24.404,21.388,-41.196
C01112=1017.426,180.451,-137.794,-24.404,21.388,-41.194
C01113=1017.425,180.851,-137.837,-24.405,21.387,-41.190
C01114=1017.423,181.252,-137.880,-24.405,21.387,-41.188
C01115=1017.422,181.654,-137.922,-24.405,21.387,-41.186
C01116=1017.422,182.054,-137.965,-24.406,21.387,-41.183
C01117=1017.421,182.455,-138.008,-24.406,21.386,-41.181
C01118=1017.420,182.856,-138.051,-24.407,21.387,-41.177
C01119=1017.419,183.257,-138.094,-24.407,21.386,-41.176
C01120=1017.417,183.657,-138.137,-24.407,21.386,-41.172
C01121=1017.417,184.059,-138.180,-24.408,21.386,-41.170
C01122=1017.415,184.459,-138.223,-24.408,21.386,-41.168
C01123=1017.415,184.860,-138.267,-24.409,21.386,-41.165
C01124=1017.414,185.262,-138.310,-24.409,21.385,-41.162
C01125=1017.413,185.662,-138.353,-24.409,21.385,-41.159
C01126=1017.411,186.064,-138.396,-24.410,21.385,-41.157
C01127=1017.410,186.464,-138.439,-24.410,21.384,-41.155
C01128=1017.409,186.866,-138.482,-24.410,21.384,-41.151
C01129=1017.408,187.267,-138.526,-24.411,21.384,-41.150
C01130=1017.407,187.668,-138.570,-24.411,21.385,-41.146
C01131=1017.406,188.068,-138.613,-24.411,21.384,-41.144
C01132=1017.405,188.469,-138.656,-24.412,21.384,-41.141
C01133=1017.405,188.871,-138.699,-24.412,21.384,-41.139
C01134=1017.404,189.272,-138.743,-24.412,21.384,-41.137
C01135=1017.403,189.673,-138.786,-24.413,21.383,-41.133
C01136=1017.402,190.074,-138.829,-24.413,21.383,-41.131
C01137=1017.401,190.475,-138.872,-24.414,21.383,-41.128
C01138=1017.400,190.876,-138.916,-24.414,21.383,-41.126
C01139=1017.399,191.278,-138.959,-24.414,21.382,-41.124
C01140=1017.398,191.678,-139.004,-24.415,21.382,-41.120
C01141=1017.398,192.079,-139.047,-24.415,21.382,-41.118
C01142=1017.397,192.481,-139.090,-24.415,21.382,-41.115
C01143=1017.396,192.882,-139.133,-24.416,21.382,-41.113
C01144=1017.395,193.283,-139.177,-24.416,21.382,-41.109
C01145=1017.395,193.684,-139.221,-24.417,21.382,-41.108
C01146=1017.393,194.085,-139.265,-24.417,21.381,-41.105
C01147=1017.393,194.486,-139.308,-24.417,21.381,-41.102
C01148=1017.392,194.888,-139.351,-24.418,21.381,-41.100
C01149=1017.391,195.288,-139.395,-24.418,21.381,-41.097
C01150=1017.391,195.689,-139.439,-24.418,21.380,-41.094
C01151=1017.389,196.091,-139.483,-24.419,21.381,-41.091
C01152=1017.389,196.491,-139.527,-24.419,21.380,-41.089
C01153=1017.388,196.893,-139.570,-24.419,21.380,-41.087
C01154=1017.388,197.293,-139.614,-24.420,21.380,-41.084
C01155=1017.387,197.695,-139.658,-24.420,21.380,-41.082
C01156=1017.386,198.097,-139.702,-24.421,21.380,-41.078
C01157=1017.386,198.497,-139.746,-24.421,21.379,-41.076
C01158=1017.385,198.899,-139.789,-24.421,21.379,-41.074
C01159=1017.384,199.297,-139.832,-24.422,21.379,-41.071
C01160=1017.383,199.686,-139.875,-24.422,21.379,-41.069
C01161=1017.383,200.087,-139.919,-24.423,21.378,-41.065
C01162=1017.383,200.299,-139.942,-24.423,21.378,-41.065
C01163=1017.382,200.522,-139.967,-24.423,21.378,-41.063
C01164=1017.382,200.752,-139.992,-24.423,21.378,-41.061
C01165=1017.381,200.979,-140.017,-24.423,21.379,-41.060
C01166=1017.381,201.386,-140.061,-24.424,21.378,-41.058
C01167=1017.380,201.737,-140.100,-24.424,21.378,-41.054
C01168=1017.381,202.086,-140.139,-24.424,21.378,-41.052
C01169=1017.382,202.473,-140.183,-24.425,21.378,-41.051
C01170=1017.388,203.689,-140.319,-24.373,21.403,-41.416
C01171=1017.390,203.938,-140.346,-24.373,21.404,-41.415
C01172=1017.392,204.186,-140.373,-24.373,21.403,-41.414
C01173=1017.393,204.435,-140.401,-24.373,21.403,-41.412
C01174=1017.395,204.683,-140.428,-24.374,21.404,-41.411
C01175=1017.397,204.932,-140.455,-24.373,21.403,-41.410
C01176=1017.399,205.180,-140.483,-24.374,21.403,-41.409
C01177=1017.401,205.430,-140.510,-24.374,21.403,-41.407
C01178=1017.403,205.678,-140.539,-24.374,21.402,-41.407
C01179=1017.405,205.926,-140.566,-24.374,21.403,-41.405
C01180=1017.407,206.175,-140.593,-24.375,21.403,-41.403
C01181=1017.409,206.423,-140.621,-24.375,21.402,-41.401
C01182=1017.411,206.672,-140.648,-24.375,21.402,-41.401
C01183=1017.413,206.920,-140.675,-24.375,21.402,-41.399
C01184=1017.414,207.168,-140.703,-24.375,21.402,-41.398
C01185=1017.416,207.417,-140.730,-24.375,21.402,-41.398
C01186=1017.419,207.665,-140.758,-24.376,21.402,-41.396
C01187=1017.421,207.914,-140.786,-24.376,21.402,-41.394
C01188=1017.423,208.163,-140.813,-24.376,21.402,-41.392
C01189=1017.425,208.405,-140.840,-24.376,21.401,-41.392
C01190=1017.426,208.647,-140.867,-24.376,21.402,-41.391
C01191=1017.428,208.891,-140.894,-24.377,21.402,-41.389
C01192=1017.431,209.133,-140.921,-24.377,21.401,-41.388
C01193=1017.433,209.376,-140.947,-24.377,21.402,-41.387
C01194=1017.434,209.618,-140.974,-24.377,21.401,-41.385
C01195=1017.436,209.861,-141.002,-24.377,21.401,-41.383
C01196=1017.438,210.104,-141.029,-24.377,21.401,-41.383
C01197=1017.440,210.352,-141.056,-24.378,21.401,-41.381
C01198=1017.442,210.601,-141.084,-24.378,21.401,-41.379
C01199=1017.444,210.849,-141.112,-24.378,21.401,-41.378
C01200=1017.447,211.098,-141.139,-24.378,21.400,-41.377
C01201=1017.448,211.346,-141.167,-24.378,21.400,-41.375
C01202=1017.450,211.595,-141.194,-24.379,21.401,-41.374
C01203=1017.453,211.842,-141.222,-24.379,21.401,-41.372
C01204=1017.455,212.092,-141.250,-24.379,21.400,-41.372
C01205=1017.457,212.340,-141.277,-24.379,21.400,-41.370
C01206=1017.459,212.588,-141.304,-24.380,21.400,-41.368
C01207=1017.461,212.837,-141.333,-24.380,21.400,-41.366
C01208=1017.464,213.085,-141.361,-24.380,21.400,-41.366
C01209=1017.465,213.334,-141.388,-24.380,21.400,-41.365
C01210=1017.467,213.582,-141.416,-24.380,21.400,-41.363
C01211=1017.469,213.830,-141.443,-24.381,21.400,-41.361
C01212=1017.472,214.079,-141.472,-24.381,21.400,-41.359
C01213=1017.474,214.327,-141.499,-24.381,21.399,-41.359
C01214=1017.476,214.576,-141.526,-24.381,21.399,-41.357
C01215=1017.478,214.825,-141.555,-24.381,21.400,-41.356
C01216=1017.481,215.072,-141.583,-24.382,21.399,-41.354
C01217=1017.483,215.316,-141.609,-24.382,21.398,-41.353
C01218=1017.484,215.558,-141.637,-24.382,21.399,-41.352
C01219=1017.487,215.801,-141.664,-24.382,21.399,-41.350
C01220=1017.489,216.043,-141.691,-24.382,21.399,-41.348
C01221=1017.491,216.287,-141.718,-24.383,21.398,-41.346
C01222=1017.493,216.529,-141.746,-24.383,21.398,-41.346
C01223=1017.495,216.772,-141.773,-24.383,21.398,-41.344
C01224=1017.497,217.014,-141.800,-24.383,21.398,-41.342
C01225=1017.500,217.263,-141.828,-24.383,21.399,-41.341
C01226=1017.502,217.512,-141.856,-24.384,21.398,-41.339
C01227=1017.505,217.760,-141.884,-24.384,21.397,-41.339
C01228=1017.506,218.009,-141.912,-24.384,21.397,-41.337
C01229=1017.509,218.257,-141.940,-24.384,21.398,-41.335
C01230=1017.511,218.506,-141.967,-24.384,21.398,-41.333
C01231=1017.513,218.754,-141.995,-24.385,21.397,-41.332
C01232=1017.516,219.003,-142.023,-24.385,21.397,-41.330
C01233=1017.518,219.250,-142.051,-24.385,21.397,-41.330
C01234=1017.520,219.499,-142.080,-24.385,21.397,-41.328
C01235=1017.523,219.747,-142.108,-24.385,21.397,-41.326
C01236=1017.525,219.996,-142.135,-24.386,21.397,-41.324
C01237=1017.529,220.371,-142.177,-24.386,21.396,-41.322
C01238=1017.532,220.745,-142.220,-24.386,21.396,-41.320
C01239=1017.536,221.121,-142.262,-24.387,21.397,-41.317
C01240=1017.539,221.495,-142.304,-24.387,21.396,-41.315
C01241=1017.542,221.744,-142.332,-24.387,21.396,-41.313
C01242=1017.544,221.992,-142.361,-24.388,21.396,-41.311
C01243=1017.547,222.241,-142.389,-24.388,21.397,-41.310
C01244=1017.549,222.488,-142.417,-24.388,21.396,-41.309
C01245=1017.552,222.848,-142.457,-24.388,21.396,-41.306
C01246=1017.555,223.208,-142.498,-24.389,21.396,-41.304
C01247=1017.559,223.567,-142.539,-24.389,21.395,-41.302
C01248=1017.562,223.926,-142.579,-24.389,21.395,-41.300
C01249=1017.565,224.175,-142.607,-24.389,21.394,-41.298
C01250=1017.567,224.423,-142.635,-24.390,21.395,-41.297
C01251=1017.570,224.672,-142.663,-24.390,21.395,-41.295
C01252=1017.573,224.920,-142.692,-24.390,21.395,-41.293
C01253=1017.574,225.168,-142.721,-24.390,21.394,-41.291
C01254=1017.577,225.417,-142.749,-24.391,21.394,-41.289
C01255=1017.580,225.665,-142.777,-24.391,21.395,-41.288
C01256=1017.582,225.913,-142.805,-24.391,21.395,-41.286
C01257=1017.585,226.162,-142.833,-24.391,21.394,-41.285
C01258=1017.587,226.410,-142.861,-24.391,21.393,-41.284
C01259=1017.590,226.659,-142.889,-24.392,21.393,-41.282
C01260=1017.593,226.907,-142.917,-24.392,21.394,-41.280
C01261=1017.594,227.156,-142.946,-24.392,21.394,-41.278
C01262=1017.597,227.404,-142.975,-24.393,21.393,-41.276
C01263=1017.600,227.652,-143.003,-24.393,21.393,-41.275
C01264=1017.602,227.900,-143.031,-24.393,21.393,-41.273
C01265=1017.605,228.149,-143.059,-24.393,21.394,-41.271
C01266=1017.608,228.398,-143.087,-24.394,21.393,-41.269
C01267=1017.610,228.646,-143.115,-24.394,21.393,-41.267
C01268=1017.613,228.894,-143.144,-24.394,21.393,-41.266
C01269=1017.615,229.137,-143.172,-24.394,21.392,-41.265
C01270=1017.617,229.380,-143.199,-24.394,21.392,-41.263
C01271=1017.620,229.623,-143.227,-24.395,21.392,-41.262
C01272=1017.623,229.867,-143.255,-24.395,21.392,-41.260
C01273=1017.625,230.109,-143.282,-24.395,21.392,-41.258
C01274=1017.628,230.352,-143.311,-24.395,21.392,-41.256
C01275=1017.630,230.595,-143.339,-24.396,21.392,-41.254
C01276=1017.633,230.838,-143.366,-24.396,21.391,-41.252
C01277=1017.636,231.086,-143.394,-24.396,21.392,-41.251
C01278=1017.638,231.335,-143.423,-24.396,21.392,-41.249
C01279=1017.641,231.583,-143.451,-24.397,21.392,-41.247
C01280=1017.643,231.832,-143.480,-24.397,21.391,-41.245
C01281=1017.646,232.079,-143.509,-24.397,21.391,-41.243
C01282=1017.649,232.328,-143.537,-24.397,21.391,-41.242
C01283=1017.651,232.577,-143.565,-24.398,21.391,-41.240
C01284=1017.655,232.825,-143.594,-24.398,21.390,-41.238
C01285=1017.658,233.073,-143.622,-24.398,21.391,-41.236
C01286=1017.660,233.322,-143.652,-24.399,21.391,-41.234
C01287=1017.662,233.570,-143.679,-24.399,21.391,-41.233
C01288=1017.665,233.818,-143.708,-24.399,21.390,-41.231
C01289=1017.668,234.066,-143.737,-24.399,21.390,-41.229
C01290=1017.671,234.315,-143.765,-24.400,21.390,-41.227
C01291=1017.673,234.563,-143.794,-24.400,21.390,-41.225
C01292=1017.676,234.812,-143.822,-24.400,21.390,-41.223
C01293=1017.679,235.060,-143.852,-24.400,21.389,-41.221
C01294=1017.682,235.309,-143.880,-24.401,21.389,-41.219
C01295=1017.685,235.557,-143.908,-24.401,21.389,-41.218
C01296=1017.687,235.805,-143.937,-24.401,21.390,-41.216
C01297=1017.690,236.048,-143.965,-24.401,21.389,-41.214
C01298=1017.692,236.291,-143.993,-24.402,21.389,-41.212
C01299=1017.695,236.534,-144.021,-24.402,21.389,-41.210
C01300=1017.698,236.777,-144.049,-24.402,21.389,-41.209
C01301=1017.701,237.020,-144.077,-24.402,21.388,-41.207
C01302=1017.704,237.264,-144.105,-24.403,21.388,-41.205
C01303=1017.706,237.507,-144.133,-24.403,21.388,-41.203
C01304=1017.709,237.750,-144.161,-24.403,21.388,-41.201
C01305=1017.712,237.998,-144.190,-24.403,21.388,-41.199
C01306=1017.715,238.246,-144.219,-24.404,21.387,-41.197
C01307=1017.718,238.495,-144.247,-24.404,21.387,-41.195
C01308=1017.720,238.743,-144.277,-24.405,21.388,-41.192
C01309=1017.723,238.992,-144.305,-24.405,21.387,-41.190
C01310=1017.727,239.240,-144.333,-24.405,21.387,-41.188
C01311=1017.729,239.488,-144.363,-24.405,21.387,-41.186
C01312=1017.732,239.736,-144.391,-24.406,21.387,-41.184
C01313=1017.735,239.985,-144.420,-24.406,21.386,-41.183
C01314=1017.738,240.233,-144.449,-24.406,21.386,-41.181
C01315=1017.742,240.481,-144.478,-24.406,21.386,-41.179
C01316=1017.744,240.730,-144.507,-24.407,21.386,-41.177
C01317=1017.747,240.978,-144.536,-24.407,21.386,-41.174
C01318=1017.750,241.227,-144.565,-24.407,21.386,-41.172
C01319=1017.753,241.474,-144.594,-24.408,21.386,-41.170
C01320=1017.756,241.723,-144.622,-24.408,21.386,-41.168
C01321=1017.758,241.971,-144.651,-24.408,21.385,-41.166
C01322=1017.762,242.219,-144.680,-24.408,21.385,-41.164
C01323=1017.764,242.468,-144.709,-24.409,21.385,-41.162
C01324=1017.768,242.716,-144.738,-24.409,21.385,-41.159
C01325=1017.770,242.960,-144.767,-24.410,21.385,-41.157
C01326=1017.774,243.202,-144.795,-24.410,21.385,-41.155
C01327=1017.776,243.446,-144.823,-24.410,21.385,-41.153
C01328=1017.780,243.689,-144.852,-24.410,21.384,-41.151
C01329=1017.782,243.932,-144.881,-24.411,21.384,-41.150
C01330=1017.785,244.175,-144.908,-24.411,21.384,-41.148
C01331=1017.788,244.418,-144.937,-24.411,21.384,-41.144
C01332=1017.791,244.662,-144.965,-24.412,21.384,-41.143
C01333=1017.794,244.911,-144.994,-24.412,21.384,-41.141
C01334=1017.797,245.159,-145.023,-24.412,21.384,-41.139
C01335=1017.800,245.407,-145.052,-24.412,21.384,-41.137
C01336=1017.803,245.656,-145.082,-24.413,21.384,-41.134
C01337=1017.807,245.903,-145.110,-24.413,21.384,-41.132
C01338=1017.809,246.152,-145.140,-24.413,21.383,-41.129
C01339=1017.813,246.400,-145.169,-24.414,21.382,-41.127
C01340=1017.816,246.649,-145.198,-24.414,21.382,-41.126
C01341=1017.819,246.897,-145.227,-24.414,21.383,-41.122
C01342=1017.822,247.145,-145.256,-24.415,21.382,-41.120
C01343=1017.825,247.393,-145.285,-24.415,21.382,-41.118
C01344=1017.829,247.642,-145.314,-24.415,21.382,-41.117
C01345=1017.831,247.889,-145.345,-24.416,21.382,-41.113
C01346=1017.835,248.137,-145.373,-24.416,21.382,-41.111
C01347=1017.838,248.386,-145.403,-24.416,21.381,-41.109
C01348=1017.841,248.634,-145.432,-24.417,21.381,-41.107
C01349=1017.844,248.882,-145.461,-24.417,21.381,-41.104
C01350=1017.847,249.131,-145.490,-24.417,21.381,-41.102
C01351=1017.851,249.379,-145.519,-24.418,21.381,-41.100
C01352=1017.853,249.627,-145.549,-24.418,21.381,-41.098
C01353=1017.857,249.871,-145.577,-24.418,21.381,-41.095
C01354=1017.860,250.114,-145.606,-24.419,21.381,-41.093
C01355=1017.863,250.357,-145.635,-24.419,21.380,-41.091
C01356=1017.867,250.601,-145.664,-24.419,21.380,-41.089
C01357=1017.870,250.844,-145.693,-24.420,21.380,-41.085
C01358=1017.873,251.087,-145.721,-24.420,21.380,-41.084
C01359=1017.876,251.331,-145.750,-24.420,21.380,-41.082
C01360=1017.879,251.575,-145.779,-24.421,21.380,-41.078
C01361=1017.883,251.822,-145.809,-24.421,21.380,-41.076
C01362=1017.886,252.070,-145.837,-24.421,21.379,-41.074
C01363=1017.889,252.319,-145.867,-24.421,21.378,-41.072
C01364=1017.892,252.567,-145.896,-24.422,21.379,-41.069
C01365=1017.896,252.815,-145.926,-24.422,21.379,-41.067
C01366=1017.899,253.063,-145.955,-24.423,21.378,-41.065
C01367=1017.902,253.312,-145.985,-24.423,21.378,-41.061
C01368=1017.906,253.560,-146.014,-24.423,21.378,-41.060
C01369=1017.909,253.809,-146.044,-24.424,21.378,-41.058
C01370=1017.912,254.056,-146.074,-24.424,21.378,-41.054
C01371=1017.915,254.305,-146.103,-24.424,21.378,-41.052
C01372=1017.919,254.553,-146.132,-24.425,21.377,-41.049
C01373=1017.922,254.801,-146.163,-24.425,21.377,-41.047
C01374=1017.925,255.049,-146.191,-24.425,21.377,-41.045
C01375=1017.929,255.298,-146.221,-24.426,21.377,-41.042
C01376=1017.932,255.546,-146.251,-24.426,21.377,-41.040
C01377=1017.936,255.794,-146.281,-24.426,21.376,-41.037
C01378=1017.939,256.042,-146.310,-24.427,21.376,-41.034
C01379=1017.943,256.290,-146.340,-24.427,21.376,-41.032
C01380=1017.946,256.539,-146.370,-24.428,21.377,-41.029
C01381=1017.949,256.783,-146.399,-24.428,21.376,-41.027
C01382=1017.953,257.026,-146.427,-24.428,21.375,-41.025
C01383=1017.956,257.270,-146.457,-24.429,21.376,-41.021
C01384=1017.959,257.512,-146.486,-24.429,21.376,-41.019
C01385=1017.962,257.756,-146.515,-24.429,21.375,-41.018
C01386=1017.966,257.999,-146.544,-24.430,21.375,-41.014
C01387=1017.970,258.243,-146.574,-24.430,21.375,-41.012
C01388=1017.987,259.479,-146.727,-24.551,21.322,-40.171
C01389=1017.989,259.759,-146.764,-24.587,21.310,-39.930
C01390=1017.992,260.038,-146.801,-24.622,21.298,-39.688
C01391=1017.994,260.318,-146.839,-24.658,21.287,-39.446
C01392=1017.995,260.597,-146.877,-24.693,21.275,-39.204
C01393=1017.996,260.845,-146.911,-24.725,21.267,-38.988
C01394=1017.996,261.092,-146.946,-24.758,21.259,-38.770
C01395=1017.996,261.340,-146.983,-24.790,21.251,-38.554
C01396=1017.996,261.587,-147.019,-24.823,21.245,-38.337
C01397=1017.994,261.867,-147.059,-24.860,21.238,-38.090
C01398=1017.994,262.146,-147.102,-24.897,21.233,-37.842
C01399=1017.992,262.426,-147.145,-24.935,21.227,-37.593
C01400=1017.990,262.705,-147.188,-24.973,21.223,-37.345
C01401=1017.988,262.952,-147.227,-25.006,21.220,-37.124
C01402=1017.986,263.199,-147.267,-25.040,21.217,-36.903
C01403=1017.983,263.445,-147.307,-25.074,21.216,-36.681
C01404=1017.979,263.693,-147.347,-25.108,21.215,-36.458
C01405=1017.975,263.972,-147.393,-25.147,21.216,-36.205
C01406=1017.970,264.250,-147.441,-25.186,21.217,-35.952
C01407=1017.965,264.530,-147.488,-25.226,21.219,-35.699
C01408=1017.960,264.809,-147.536,-25.265,21.221,-35.444
C01409=1017.954,265.055,-147.580,-25.300,21.225,-35.219
C01410=1017.949,265.301,-147.623,-25.335,21.229,-34.991
C01411=1017.943,265.548,-147.668,-25.370,21.233,-34.766
C01412=1017.936,265.793,-147.712,-25.406,21.239,-34.538
C01413=1017.929,266.072,-147.764,-25.446,21.246,-34.279
C01414=1017.921,266.351,-147.816,-25.487,21.254,-34.021
C01415=1017.912,266.630,-147.868,-25.527,21.264,-33.760
C01416=1017.903,266.908,-147.922,-25.568,21.275,-33.499
C01417=1017.895,267.153,-147.970,-25.604,21.284,-33.269
C01418=1017.886,267.398,-148.018,-25.641,21.295,-33.037
C01419=1017.877,267.644,-148.067,-25.677,21.306,-32.805
C01420=1017.867,267.889,-148.116,-25.713,21.318,-32.573
C01421=1017.857,268.168,-148.172,-25.755,21.333,-32.307
C01422=1017.845,268.447,-148.230,-25.797,21.350,-32.039
C01423=1017.833,268.725,-148.288,-25.839,21.367,-31.772
C01424=1017.820,269.004,-148.346,-25.881,21.386,-31.502
C01425=1017.809,269.248,-148.398,-25.918,21.402,-31.266
C01426=1017.797,269.492,-148.451,-25.955,21.420,-31.029
C01427=1017.785,269.736,-148.504,-25.992,21.439,-30.791
C01428=1017.772,269.980,-148.558,-26.030,21.459,-30.551
C01429=1017.758,270.259,-148.619,-26.072,21.483,-30.277
C01430=1017.742,270.536,-148.682,-26.115,21.507,-30.003
C01431=1017.726,270.815,-148.744,-26.158,21.533,-29.728
C01432=1017.710,271.093,-148.809,-26.201,21.560,-29.450
C01433=1017.695,271.336,-148.865,-26.238,21.585,-29.208
C01434=1017.681,271.580,-148.921,-26.276,21.610,-28.964
C01435=1017.665,271.823,-148.979,-26.314,21.637,-28.720
C01436=1017.649,272.065,-149.036,-26.351,21.664,-28.476
C01437=1017.631,272.344,-149.104,-26.395,21.697,-28.194
C01438=1017.612,272.622,-149.172,-26.438,21.731,-27.910
C01439=1017.592,272.899,-149.240,-26.481,21.766,-27.626
C01440=1017.573,273.177,-149.309,-26.525,21.803,-27.342
C01441=1017.555,273.419,-149.370,-26.562,21.835,-27.092
C01442=1017.537,273.661,-149.432,-26.600,21.869,-26.841
C01443=1017.518,273.902,-149.493,-26.638,21.903,-26.590
C01444=1017.500,274.144,-149.556,-26.676,21.940,-26.336
C01445=1017.477,274.422,-149.627,-26.720,21.983,-26.043
C01446=1017.455,274.700,-149.701,-26.763,22.027,-25.750
C01447=1017.432,274.977,-149.775,-26.807,22.073,-25.453
C01448=1017.408,275.254,-149.849,-26.851,22.119,-25.156
C01449=1017.387,275.495,-149.914,-26.889,22.162,-24.896
C01450=1017.366,275.735,-149.980,-26.927,22.204,-24.635
C01451=1017.343,275.975,-150.047,-26.965,22.250,-24.373
C01452=1017.321,276.216,-150.113,-27.003,22.294,-24.111
C01453=1017.295,276.493,-150.192,-27.046,22.349,-23.804
C01454=1017.269,276.770,-150.270,-27.090,22.404,-23.496
C01455=1017.242,277.047,-150.349,-27.134,22.462,-23.186
C01456=1017.214,277.324,-150.430,-27.177,22.521,-22.877
C01457=1017.190,277.563,-150.499,-27.215,22.573,-22.606
C01458=1017.165,277.802,-150.569,-27.252,22.626,-22.334
C01459=1017.140,278.041,-150.640,-27.290,22.681,-22.062
C01460=1017.115,278.279,-150.712,-27.327,22.737,-21.789
C01461=1017.085,278.556,-150.796,-27.370,22.804,-21.469
C01462=1017.054,278.833,-150.880,-27.413,22.873,-21.147
C01463=1017.023,279.109,-150.965,-27.456,22.942,-20.824
C01464=1016.992,279.386,-151.051,-27.498,23.014,-20.499
C01465=1016.964,279.622,-151.125,-27.534,23.078,-20.218
C01466=1016.936,279.859,-151.199,-27.570,23.142,-19.936
C01467=1016.907,280.096,-151.275,-27.606,23.208,-19.653
C01468=1016.879,280.333,-151.351,-27.642,23.276,-19.367
C01469=1016.845,280.610,-151.441,-27.684,23.357,-19.031
C01470=1016.810,280.885,-151.531,-27.725,23.440,-18.691
C01471=1016.775,281.161,-151.622,-27.766,23.526,-18.349
C01472=1016.739,281.436,-151.713,-27.807,23.613,-18.004
C01473=1016.708,281.672,-151.793,-27.842,23.690,-17.706
C01474=1016.677,281.906,-151.872,-27.877,23.768,-17.406
C01475=1016.645,282.142,-151.952,-27.911,23.848,-17.104
C01476=1016.612,282.376,-152.033,-27.945,23.929,-16.801
C01477=1016.574,282.651,-152.128,-27.984,24.027,-16.441
C01478=1016.535,282.926,-152.225,-28.023,24.128,-16.079
C01479=1016.495,283.201,-152.321,-28.062,24.232,-15.713
C01480=1016.456,283.476,-152.420,-28.100,24.338,-15.343
C01481=1016.421,283.709,-152.504,-28.132,24.429,-15.026
C01482=1016.386,283.941,-152.588,-28.164,24.524,-14.708
C01483=1016.351,284.174,-152.673,-28.195,24.619,-14.388
C01484=1016.314,284.407,-152.759,-28.226,24.716,-14.065
C01485=1016.272,284.681,-152.861,-28.261,24.835,-13.680
C01486=1016.229,284.955,-152.963,-28.296,24.955,-13.292
C01487=1016.184,285.228,-153.067,-28.330,25.079,-12.901
C01488=1016.140,285.502,-153.171,-28.364,25.204,-12.507
C01489=1016.102,285.732,-153.260,-28.391,25.314,-12.171
C01490=1016.062,285.962,-153.350,-28.418,25.425,-11.832
C01491=1016.024,286.193,-153.440,-28.444,25.537,-11.492
C01492=1015.984,286.423,-153.530,-28.470,25.652,-11.148
C01493=1015.937,286.695,-153.638,-28.499,25.792,-10.737
C01494=1015.889,286.968,-153.748,-28.527,25.936,-10.320
C01495=1015.839,287.240,-153.858,-28.555,26.082,-9.899
C01496=1015.790,287.512,-153.969,-28.581,26.233,-9.471
C01497=1015.748,287.740,-154.063,-28.602,26.363,-9.109
C01498=1015.705,287.968,-154.158,-28.622,26.495,-8.743
C01499=1015.662,288.195,-154.253,-28.641,26.630,-8.372
C01500=1015.619,288.422,-154.349,-28.659,26.767,-7.999
C01501=1015.567,288.694,-154.465,-28.679,26.937,-7.545
C01502=1015.513,288.964,-154.581,-28.698,27.109,-7.088
C01503=1015.460,289.236,-154.698,-28.715,27.285,-6.624
C01504=1015.405,289.505,-154.816,-28.730,27.467,-6.153
C01505=1015.359,289.729,-154.916,-28.742,27.622,-5.757
C01506=1015.312,289.954,-155.016,-28.752,27.779,-5.357
C01507=1015.265,290.178,-155.116,-28.760,27.939,-4.952
C01508=1015.218,290.402,-155.217,-28.767,28.103,-4.544
C01509=1015.160,290.672,-155.340,-28.773,28.305,-4.046
C01510=1015.101,290.941,-155.464,-28.777,28.512,-3.541
C01511=1015.043,291.208,-155.589,-28.778,28.722,-3.030
C01512=1014.982,291.477,-155.714,-28.777,28.937,-2.514
C01513=1014.933,291.698,-155.819,-28.773,29.120,-2.080
C01514=1014.881,291.919,-155.925,-28.768,29.306,-1.642
C01515=1014.831,292.140,-156.031,-28.760,29.494,-1.200
C01516=1014.779,292.361,-156.139,-28.751,29.686,-0.753
C01517=1014.715,292.627,-156.269,-28.736,29.926,-0.203
C01518=1014.652,292.894,-156.400,-28.717,30.168,0.353
C01519=1014.587,293.159,-156.534,-28.695,30.417,0.916
C01520=1014.521,293.424,-156.667,-28.669,30.673,1.490
C01521=1014.466,293.642,-156.778,-28.645,30.886,1.967
C01522=1014.411,293.859,-156.890,-28.617,31.104,2.450
C01523=1014.355,294.075,-157.002,-28.586,31.327,2.940
C01524=1014.299,294.292,-157.115,-28.552,31.552,3.436
C01525=1014.230,294.555,-157.254,-28.506,31.835,4.050
C01526=1014.160,294.819,-157.393,-28.455,32.123,4.674
C01527=1014.089,295.081,-157.535,-28.398,32.417,5.306
C01528=1014.018,295.344,-157.677,-28.335,32.716,5.947
C01529=1013.958,295.557,-157.795,-28.280,32.966,6.479
C01530=1013.899,295.770,-157.912,-28.220,33.220,7.016
C01531=1013.838,295.981,-158.030,-28.156,33.478,7.560
C01532=1013.777,296.193,-158.150,-28.087,33.740,8.111
C01533=1013.701,296.453,-158.298,-27.996,34.069,8.801
C01534=1013.625,296.713,-158.447,-27.897,34.404,9.500
C01535=1013.548,296.972,-158.596,-27.790,34.746,10.213
C01536=1013.469,297.230,-158.748,-27.675,35.094,10.935
C01537=1013.405,297.438,-158.871,-27.576,35.380,11.529
C01538=1013.341,297.646,-158.995,-27.470,35.670,12.129
C01539=1013.277,297.853,-159.120,-27.359,35.964,12.737
C01540=1013.211,298.060,-159.246,-27.241,36.263,13.354
C01541=1013.128,298.316,-159.402,-27.085,36.640,14.133
C01542=1013.044,298.572,-159.561,-26.918,37.024,14.926
C01543=1012.961,298.826,-159.720,-26.741,37.414,15.733
C01544=1012.876,299.081,-159.881,-26.551,37.810,16.553
C01545=1012.807,299.283,-160.011,-26.391,38.132,17.220
C01546=1012.737,299.485,-160.141,-26.221,38.458,17.898
C01547=1012.667,299.686,-160.272,-26.044,38.788,18.586
C01548=1012.597,299.888,-160.404,-25.857,39.121,19.283
///RCONF 0,0,0,0,0,0,0,0,0,0,0,0,0,0,0,0,0,0,0,0,0,0,0,0
C01549=1012.507,300.139,-160.571,-25.611,39.544,20.170
C01550=1012.416,300.390,-160.739,-25.349,39.974,21.077
C01551=1012.325,300.639,-160.909,-25.071,40.409,21.999
C01552=1012.232,300.888,-161.079,-24.778,40.847,22.938
C01553=1012.159,301.084,-161.216,-24.533,41.199,23.695
C01554=1012.084,301.280,-161.353,-24.278,41.553,24.463
C01555=1012.009,301.475,-161.490,-24.011,41.910,25.243
C01556=1011.933,301.670,-161.629,-23.731,42.271,26.037
C01557=1011.837,301.916,-161.806,-23.359,42.732,27.060
C01558=1011.739,302.161,-161.984,-22.967,43.196,28.105
C01559=1011.639,302.405,-162.163,-22.552,43.665,29.173
C01560=1011.540,302.648,-162.345,-22.115,44.137,30.264
C01561=1011.461,302.838,-162.487,-21.757,44.508,31.133
C01562=1011.381,303.026,-162.630,-21.384,44.880,32.017
C01563=1011.301,303.215,-162.775,-20.997,45.253,32.914
C01564=1011.220,303.402,-162.920,-20.593,45.627,33.826
C01565=1011.115,303.642,-163.107,-20.052,46.107,35.019
C01566=1011.010,303.880,-163.296,-19.485,46.587,36.235
C01567=1010.903,304.118,-163.486,-18.890,47.066,37.479
C01568=1010.795,304.354,-163.677,-18.265,47.545,38.750
C01569=1010.710,304.536,-163.826,-17.761,47.914,39.754
C01570=1010.626,304.718,-163.976,-17.237,48.283,40.777
C01571=1010.541,304.899,-164.127,-16.695,48.650,41.816
C01572=1010.455,305.079,-164.278,-16.132,49.015,42.875
C01573=1010.342,305.311,-164.476,-15.372,49.485,44.275
C01574=1010.228,305.543,-164.675,-14.580,49.949,45.706
C01575=1010.114,305.772,-164.875,-13.751,50.408,47.169
C01576=1009.998,306.001,-165.077,-12.888,50.859,48.662
C01577=1009.909,306.175,-165.232,-12.202,51.199,49.829
C01578=1009.819,306.349,-165.388,-11.496,51.534,51.012
C01579=1009.728,306.521,-165.545,-10.767,51.863,52.216
C01580=1009.637,306.694,-165.703,-10.018,52.186,53.439
C01581=1009.517,306.918,-165.911,-9.002,52.599,55.068
C01582=1009.397,307.141,-166.120,-7.948,53.000,56.733
C01583=1009.273,307.363,-166.330,-6.854,53.388,58.434
C01584=1009.150,307.582,-166.542,-5.724,53.761,60.165
C01585=1009.056,307.748,-166.703,-4.837,54.035,61.506
C01586=1008.962,307.914,-166.865,-3.930,54.299,62.863
C01587=1008.865,308.078,-167.028,-2.999,54.554,64.242
C01588=1008.769,308.242,-167.192,-2.047,54.798,65.640
C01589=1008.641,308.457,-167.409,-0.758,55.103,67.512
C01590=1008.513,308.670,-167.628,0.564,55.388,69.411
C01591=1008.383,308.882,-167.848,1.921,55.651,71.337
C01592=1008.252,309.093,-168.069,3.305,55.891,73.285
C01593=1008.094,309.343,-168.335,5.000,56.149,75.646
C01594=1007.928,309.590,-168.598,6.734,56.371,78.036
C01595=1007.742,309.832,-168.850,8.495,56.557,80.442
C01596=1007.539,310.068,-169.090,10.267,56.705,82.842
C01597=1007.846,310.192,-169.430,10.995,56.755,83.823
C01598=1007.963,310.064,-169.302,10.016,56.687,82.503
C01599=1008.074,309.933,-169.171,9.038,56.607,81.179
C01600=1008.182,309.802,-169.034,8.063,56.515,79.854
C01601=1008.284,309.668,-168.896,7.094,56.413,78.529
C01602=1008.380,309.533,-168.753,6.129,56.298,77.205
C01603=1008.471,309.396,-168.607,5.176,56.173,75.889
C01604=1008.558,309.259,-168.461,4.234,56.037,74.582
C01605=1008.645,309.121,-168.314,3.305,55.891,73.285
C01606=1008.776,308.910,-168.093,1.921,55.651,71.337
C01607=1008.905,308.699,-167.873,0.564,55.388,69.411
C01608=1009.035,308.485,-167.655,-0.758,55.103,67.512
C01609=1009.162,308.270,-167.437,-2.047,54.798,65.640
C01610=1009.259,308.106,-167.274,-2.999,54.554,64.242
C01611=1009.354,307.942,-167.111,-3.930,54.299,62.863
C01612=1009.449,307.777,-166.948,-4.837,54.035,61.506
C01613=1009.543,307.611,-166.787,-5.724,53.761,60.165
C01614=1009.666,307.390,-166.575,-6.854,53.388,58.434
C01615=1009.789,307.169,-166.365,-7.948,53.000,56.733
C01616=1009.910,306.946,-166.155,-9.002,52.599,55.068
C01617=1010.031,306.722,-165.948,-10.018,52.186,53.439
C01618=1010.121,306.550,-165.791,-10.767,51.863,52.216
C01619=1010.212,306.377,-165.634,-11.496,51.534,51.012
C01620=1010.303,306.203,-165.477,-12.202,51.199,49.829
C01621=1010.391,306.029,-165.321,-12.888,50.859,48.662
C01622=1010.507,305.801,-165.120,-13.751,50.408,47.169
C01623=1010.621,305.571,-164.919,-14.578,49.950,45.708
C01624=1010.735,305.340,-164.721,-15.372,49.485,44.275
C01625=1010.847,305.107,-164.523,-16.132,49.015,42.875
C01626=1010.933,304.927,-164.372,-16.695,48.650,41.816
C01627=1011.019,304.746,-164.221,-17.237,48.283,40.777
C01628=1011.104,304.565,-164.071,-17.761,47.914,39.754
C01629=1011.187,304.383,-163.922,-18.265,47.545,38.750
C01630=1011.295,304.146,-163.731,-18.890,47.066,37.479
C01631=1011.402,303.909,-163.541,-19.485,46.587,36.235
C01632=1011.508,303.671,-163.352,-20.052,46.107,35.019
C01633=1011.612,303.430,-163.165,-20.593,45.627,33.826
C01634=1011.694,303.243,-163.020,-20.997,45.253,32.914
C01635=1011.773,303.055,-162.875,-21.384,44.880,32.017
C01636=1011.853,302.866,-162.732,-21.757,44.508,31.133
C01637=1011.932,302.676,-162.590,-22.115,44.137,30.264
C01638=1012.033,302.433,-162.409,-22.552,43.665,29.173
C01639=1012.131,302.189,-162.229,-22.967,43.196,28.105
C01640=1012.229,301.944,-162.051,-23.359,42.732,27.060
C01641=1012.327,301.699,-161.874,-23.731,42.271,26.037
C01642=1012.402,301.504,-161.735,-24.011,41.910,25.243
C01643=1012.477,301.309,-161.597,-24.278,41.553,24.463
C01644=1012.551,301.113,-161.461,-24.533,41.199,23.695
C01645=1012.626,300.917,-161.324,-24.778,40.847,22.938
C01646=1012.718,300.668,-161.154,-25.071,40.409,21.999
C01647=1012.810,300.417,-160.984,-25.349,39.974,21.077
C01648=1012.900,300.168,-160.816,-25.611,39.544,20.170
///RCONF 0,0,0,0,1,0,0,0,0,0,0,0,0,0,0,0,0,0,0,0,0,0,0,0
C01649=1012.990,299.916,-160.649,-25.857,39.121,19.283
C01650=1013.060,299.715,-160.517,-26.044,38.788,18.586
C01651=1013.130,299.513,-160.386,-26.221,38.458,17.898
C01652=1013.199,299.311,-160.255,-26.391,38.132,17.220
C01653=1013.268,299.109,-160.126,-26.551,37.810,16.553
C01654=1013.353,298.855,-159.965,-26.741,37.414,15.733
C01655=1013.438,298.601,-159.805,-26.918,37.024,14.926
C01656=1013.521,298.345,-159.647,-27.085,36.640,14.133
C01657=1013.603,298.088,-159.490,-27.241,36.263,13.354
C01658=1013.669,297.881,-159.365,-27.359,35.964,12.737
C01659=1013.734,297.674,-159.240,-27.470,35.670,12.129
C01660=1013.799,297.467,-159.116,-27.576,35.380,11.529
C01661=1013.862,297.259,-158.993,-27.675,35.094,10.935
C01662=1013.941,297.000,-158.841,-27.790,34.746,10.213
C01663=1014.018,296.742,-158.691,-27.897,34.404,9.500
C01664=1014.095,296.482,-158.542,-27.996,34.069,8.801
C01665=1014.171,296.222,-158.395,-28.087,33.740,8.111
C01666=1014.231,296.010,-158.275,-28.156,33.478,7.560
C01667=1014.291,295.798,-158.157,-28.220,33.220,7.016
C01668=1014.351,295.585,-158.039,-28.280,32.966,6.479
C01669=1014.410,295.372,-157.922,-28.335,32.716,5.947
C01670=1014.482,295.110,-157.780,-28.398,32.417,5.306
C01671=1014.553,294.848,-157.640,-28.455,32.123,4.674
C01672=1014.623,294.585,-157.499,-28.506,31.835,4.050
C01673=1014.693,294.320,-157.360,-28.552,31.552,3.436
C01674=1014.749,294.104,-157.247,-28.586,31.327,2.940
C01675=1014.804,293.887,-157.135,-28.617,31.104,2.450
C01676=1014.859,293.670,-157.023,-28.645,30.886,1.967
C01677=1014.914,293.453,-156.913,-28.669,30.673,1.490
C01678=1014.979,293.187,-156.779,-28.695,30.417,0.916
C01679=1015.044,292.921,-156.646,-28.717,30.168,0.353
C01680=1015.108,292.656,-156.514,-28.736,29.926,-0.203
C01681=1015.172,292.388,-156.384,-28.751,29.686,-0.753
C01682=1015.223,292.169,-156.277,-28.760,29.494,-1.200
C01683=1015.274,291.948,-156.170,-28.768,29.306,-1.642
C01684=1015.325,291.727,-156.065,-28.773,29.120,-2.080
C01685=1015.376,291.505,-155.960,-28.777,28.937,-2.514
C01686=1015.435,291.238,-155.834,-28.778,28.722,-3.030
C01687=1015.495,290.970,-155.709,-28.777,28.512,-3.541
C01688=1015.553,290.700,-155.585,-28.773,28.305,-4.046
C01689=1015.611,290.431,-155.462,-28.767,28.103,-4.544
C01690=1015.659,290.207,-155.361,-28.760,27.939,-4.952
C01691=1015.705,289.983,-155.260,-28.752,27.779,-5.357
C01692=1015.752,289.758,-155.161,-28.742,27.622,-5.757
C01693=1015.798,289.533,-155.061,-28.730,27.467,-6.153
C01694=1015.853,289.263,-154.943,-28.715,27.285,-6.624
C01695=1015.907,288.993,-154.826,-28.698,27.109,-7.088
C01696=1015.959,288.722,-154.709,-28.679,26.937,-7.545
C01697=1016.012,288.451,-154.594,-28.659,26.767,-7.999
C01698=1016.055,288.223,-154.498,-28.641,26.630,-8.372
C01699=1016.098,287.996,-154.403,-28.622,26.495,-8.743
C01700=1016.141,287.769,-154.308,-28.602,26.363,-9.109
C01701=1016.183,287.540,-154.214,-28.581,26.233,-9.471
C01702=1016.232,287.269,-154.103,-28.555,26.082,-9.899
C01703=1016.281,286.997,-153.992,-28.527,25.936,-10.320
C01704=1016.329,286.724,-153.884,-28.499,25.792,-10.737
C01705=1016.376,286.451,-153.775,-28.470,25.652,-11.148
C01706=1016.416,286.221,-153.684,-28.444,25.537,-11.492
C01707=1016.456,285.991,-153.595,-28.418,25.425,-11.832
C01708=1016.494,285.761,-153.504,-28.391,25.314,-12.171
C01709=1016.532,285.530,-153.415,-28.364,25.204,-12.507
C01710=1016.577,285.256,-153.312,-28.330,25.079,-12.901
C01711=1016.621,284.983,-153.208,-28.296,24.955,-13.292
C01712=1016.664,284.709,-153.106,-28.261,24.835,-13.680
C01713=1016.708,284.435,-153.004,-28.226,24.716,-14.065
C01714=1016.743,284.202,-152.918,-28.195,24.619,-14.388
C01715=1016.779,283.970,-152.833,-28.164,24.524,-14.708
C01716=1016.814,283.737,-152.748,-28.132,24.429,-15.026
C01717=1016.848,283.504,-152.664,-28.100,24.338,-15.343
C01718=1016.888,283.230,-152.567,-28.062,24.232,-15.713
C01719=1016.928,282.954,-152.470,-28.023,24.128,-16.079
C01720=1016.967,282.680,-152.373,-27.984,24.027,-16.441
C01721=1017.006,282.405,-152.278,-27.945,23.929,-16.801
C01722=1017.037,282.170,-152.197,-27.911,23.848,-17.104
C01723=1017.069,281.935,-152.117,-27.877,23.768,-17.406
C01724=1017.100,281.700,-152.037,-27.842,23.690,-17.706
C01725=1017.131,281.464,-151.958,-27.807,23.613,-18.004
C01726=1017.167,281.189,-151.867,-27.766,23.526,-18.349
C01727=1017.203,280.913,-151.775,-27.725,23.440,-18.691
C01728=1017.237,280.638,-151.685,-27.684,23.357,-19.031
C01729=1017.271,280.362,-151.596,-27.642,23.276,-19.367
C01730=1017.301,280.125,-151.520,-27.606,23.208,-19.653
C01731=1017.328,279.888,-151.444,-27.570,23.142,-19.936
C01732=1017.356,279.651,-151.370,-27.534,23.078,-20.218
C01733=1017.384,279.414,-151.295,-27.498,23.014,-20.499
C01734=1017.416,279.138,-151.209,-27.456,22.942,-20.824
C01735=1017.447,278.861,-151.124,-27.413,22.873,-21.147
C01736=1017.478,278.584,-151.040,-27.370,22.804,-21.469
C01737=1017.508,278.307,-150.957,-27.327,22.737,-21.789
C01738=1017.532,278.069,-150.885,-27.290,22.681,-22.062
C01739=1017.557,277.830,-150.814,-27.252,22.626,-22.334
C01740=1017.582,277.591,-150.744,-27.215,22.573,-22.606
C01741=1017.607,277.352,-150.674,-27.177,22.521,-22.877
C01742=1017.634,277.075,-150.594,-27.134,22.462,-23.186
C01743=1017.661,276.798,-150.515,-27.090,22.404,-23.496
C01744=1017.688,276.521,-150.436,-27.046,22.349,-23.804
C01745=1017.714,276.244,-150.358,-27.003,22.295,-24.109
C01746=1017.736,276.003,-150.291,-26.965,22.250,-24.373
C01747=1017.758,275.764,-150.225,-26.927,22.204,-24.635
C01748=1017.779,275.524,-150.159,-26.889,22.162,-24.896
C01749=1017.800,275.283,-150.094,-26.851,22.119,-25.156
C01750=1017.824,275.006,-150.019,-26.807,22.073,-25.453
C01751=1017.847,274.728,-149.945,-26.763,22.027,-25.750
C01752=1017.869,274.450,-149.872,-26.720,21.983,-26.043
C01753=1017.892,274.172,-149.800,-26.676,21.940,-26.336
C01754=1017.911,273.931,-149.738,-26.638,21.903,-26.590
C01755=1017.930,273.689,-149.676,-26.600,21.869,-26.841
C01756=1017.947,273.447,-149.614,-26.562,21.835,-27.092
C01757=1017.966,273.206,-149.554,-26.525,21.803,-27.342
C01758=1017.985,272.927,-149.485,-26.481,21.766,-27.626
C01759=1018.004,272.650,-149.416,-26.438,21.731,-27.910
C01760=1018.024,272.372,-149.349,-26.395,21.697,-28.194
C01761=1018.041,272.094,-149.281,-26.351,21.664,-28.476
C01762=1018.058,271.851,-149.224,-26.314,21.637,-28.720
C01763=1018.073,271.608,-149.166,-26.276,21.610,-28.964
C01764=1018.088,271.365,-149.110,-26.238,21.585,-29.208
C01765=1018.102,271.122,-149.053,-26.201,21.560,-29.450
C01766=1018.119,270.843,-148.989,-26.158,21.533,-29.728
C01767=1018.134,270.565,-148.925,-26.115,21.507,-30.003
C01768=1018.150,270.287,-148.864,-26.072,21.483,-30.277
C01769=1018.165,270.009,-148.802,-26.030,21.459,-30.551
C01770=1018.177,269.764,-148.748,-25.992,21.439,-30.791
C01771=1018.189,269.520,-148.696,-25.955,21.420,-31.029
C01772=1018.201,269.276,-148.643,-25.918,21.402,-31.266
C01773=1018.213,269.032,-148.591,-25.881,21.386,-31.502
C01774=1018.225,268.753,-148.533,-25.839,21.367,-31.772
C01775=1018.237,268.475,-148.475,-25.797,21.350,-32.039
C01776=1018.249,268.196,-148.417,-25.755,21.333,-32.307
C01777=1018.260,267.918,-148.361,-25.714,21.319,-32.571
C01778=1018.270,267.673,-148.311,-25.677,21.306,-32.805
C01779=1018.279,267.427,-148.262,-25.641,21.295,-33.037
C01780=1018.287,267.182,-148.215,-25.604,21.284,-33.269
C01781=1018.296,266.937,-148.167,-25.568,21.275,-33.499
C01782=1018.304,266.658,-148.113,-25.527,21.264,-33.760
C01783=1018.313,266.379,-148.061,-25.487,21.254,-34.021
